      A     M    502.5;
      =     L      0.0;
      BLD   103;
      A     I    304.4;
      =     L      0.1;
      BLD   103;
      A     I    304.5;
      =     L      0.2;
      BLD   103;
      A     I    304.6;
      =     L      0.4;
      BLD   103;
      A     I    304.7;
      =     L      0.6;
      BLD   103;
      A     I    305.0;
      =     L      1.0;
      BLD   103;
      A     I    305.1;
      =     L      1.2;
      BLD   103;
      A     M    740.6;
      =     L      2.1;
      BLD   103;
      A     M    740.7;
      =     L      2.2;
      BLD   103;
      AN    M    504.0;
      AN    M    504.1;
      AN    M   6060.0;
      AN    M   6260.0;
      AN    M   6280.0;
      AN    M    504.2;
      A     M    500.2;
      =     L      2.3;
      BLD   103;
      A(    ;
      O     I      0.1;
      O     M   4120.1;
      )     ;
      =     L      2.5;
      BLD   103;
      A     M      0.5;
      =     L      2.6;
      BLD   103;
      CALL #S705_TL_DC_1ST_CLAMP1 (
           Enable_Aux               := L      0.0,
           Adv_Amount               := 1,
           Ret_Amount               := 5,
           LS_Adv1                  := L      0.1,
           LS_Ret1                  := L      0.2,
           LS_Ret2                  := L      0.4,
           LS_Ret3                  := L      0.6,
           LS_Ret4                  := L      1.0,
           LS_Ret5                  := L      1.2,
           SOL_Adv                  := L      2.1,
           SOL_Ret                  := L      2.2,
           M_Ready                  := L      2.3,
           T_CHK1                   := T#4S,
           T_CHK2                   := T#4S,
           PB_Error_Rst             := L      2.5,
           M_FLICK                  := L      2.6,
           M_Adv_Err                := M    750.6,
           M_Ret_Err                := M    750.7,
           Visu_Adv                 := DB51.DBW  132,
           Visu_Ret                 := DB51.DBW  134);
      NOP   0;
NETWORK
TITLE =
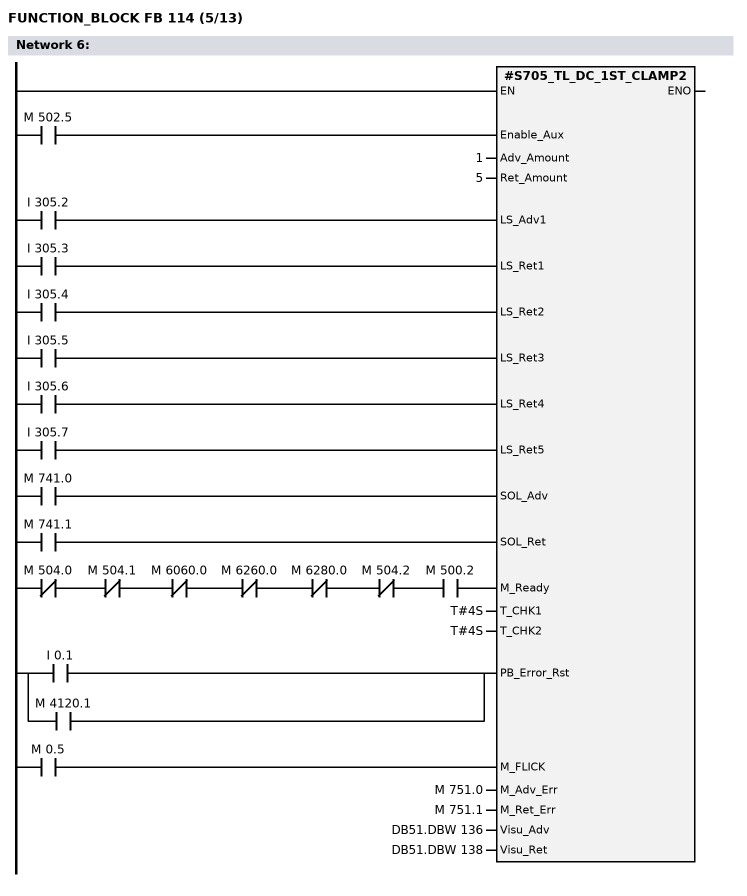

      A     M    502.5;
      =     L      0.0;
      BLD   103;
      A     I    305.2;
      =     L      0.1;
      BLD   103;
      A     I    305.3;
      =     L      0.2;
      BLD   103;
      A     I    305.4;
      =     L      0.4;
      BLD   103;
      A     I    305.5;
      =     L      0.6;
      BLD   103;
      A     I    305.6;
      =     L      1.0;
      BLD   103;
      A     I    305.7;
      =     L      1.2;
      BLD   103;
      A     M    741.0;
      =     L      2.1;
      BLD   103;
      A     M    741.1;
      =     L      2.2;
      BLD   103;
      AN    M    504.0;
      AN    M    504.1;
      AN    M   6060.0;
      AN    M   6260.0;
      AN    M   6280.0;
      AN    M    504.2;
      A     M    500.2;
      =     L      2.3;
      BLD   103;
      A(    ;
      O     I      0.1;
      O     M   4120.1;
      )     ;
      =     L      2.5;
      BLD   103;
      A     M      0.5;
      =     L      2.6;
      BLD   103;
      CALL #S705_TL_DC_1ST_CLAMP2 (
           Enable_Aux               := L      0.0,
           Adv_Amount               := 1,
           Ret_Amount               := 5,
           LS_Adv1                  := L      0.1,
           LS_Ret1                  := L      0.2,
           LS_Ret2                  := L      0.4,
           LS_Ret3                  := L      0.6,
           LS_Ret4                  := L      1.0,
           LS_Ret5                  := L      1.2,
           SOL_Adv                  := L      2.1,
           SOL_Ret                  := L      2.2,
           M_Ready                  := L      2.3,
           T_CHK1                   := T#4S,
           T_CHK2                   := T#4S,
           PB_Error_Rst             := L      2.5,
           M_FLICK                  := L      2.6,
           M_Adv_Err                := M    751.0,
           M_Ret_Err                := M    751.1,
           Visu_Adv                 := DB51.DBW  136,
           Visu_Ret                 := DB51.DBW  138);
      NOP   0;
NETWORK
TITLE =
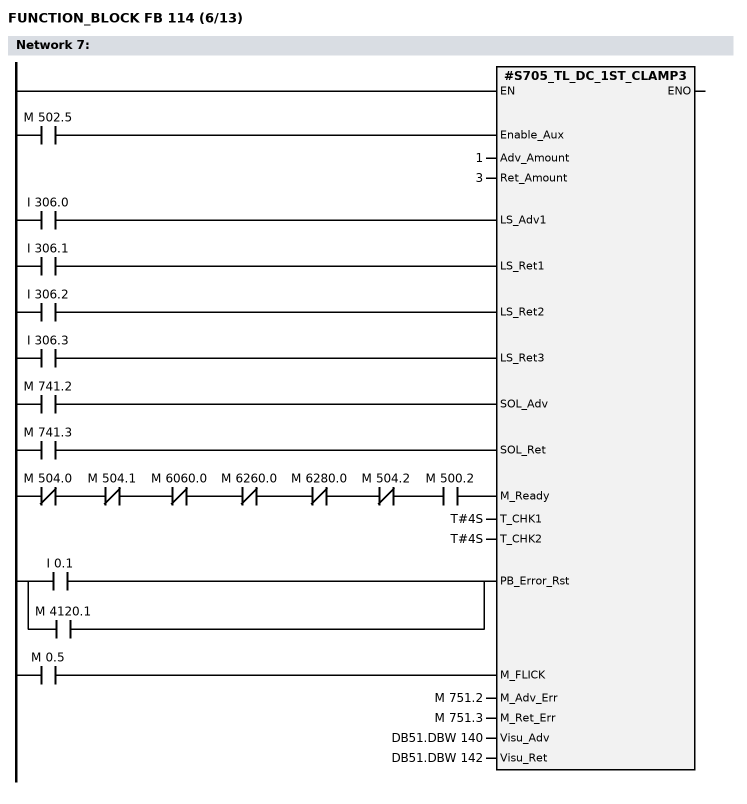

      A     M    502.5;
      =     L      0.0;
      BLD   103;
      A     I    306.0;
      =     L      0.1;
      BLD   103;
      A     I    306.1;
      =     L      0.2;
      BLD   103;
      A     I    306.2;
      =     L      0.4;
      BLD   103;
      A     I    306.3;
      =     L      0.6;
      BLD   103;
      A     M    741.2;
      =     L      2.1;
      BLD   103;
      A     M    741.3;
      =     L      2.2;
      BLD   103;
      AN    M    504.0;
      AN    M    504.1;
      AN    M   6060.0;
      AN    M   6260.0;
      AN    M   6280.0;
      AN    M    504.2;
      A     M    500.2;
      =     L      2.3;
      BLD   103;
      A(    ;
      O     I      0.1;
      O     M   4120.1;
      )     ;
      =     L      2.5;
      BLD   103;
      A     M      0.5;
      =     L      2.6;
      BLD   103;
      CALL #S705_TL_DC_1ST_CLAMP3 (
           Enable_Aux               := L      0.0,
           Adv_Amount               := 1,
           Ret_Amount               := 3,
           LS_Adv1                  := L      0.1,
           LS_Ret1                  := L      0.2,
           LS_Ret2                  := L      0.4,
           LS_Ret3                  := L      0.6,
           SOL_Adv                  := L      2.1,
           SOL_Ret                  := L      2.2,
           M_Ready                  := L      2.3,
           T_CHK1                   := T#4S,
           T_CHK2                   := T#4S,
           PB_Error_Rst             := L      2.5,
           M_FLICK                  := L      2.6,
           M_Adv_Err                := M    751.2,
           M_Ret_Err                := M    751.3,
           Visu_Adv                 := DB51.DBW  140,
           Visu_Ret                 := DB51.DBW  142);
      NOP   0;
NETWORK
TITLE =
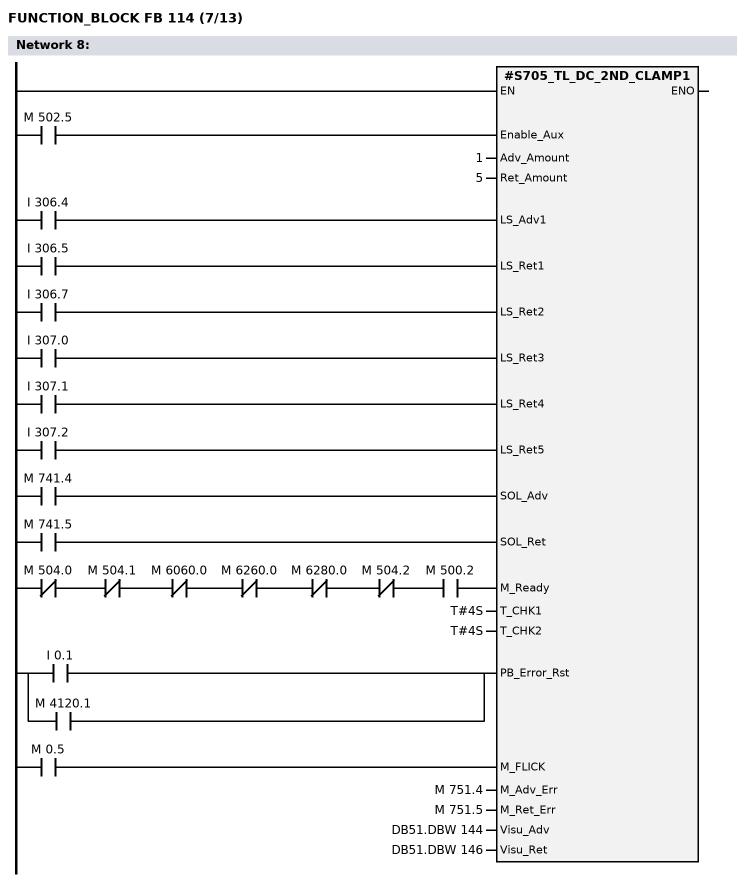

      A     M    502.5;
      =     L      0.0;
      BLD   103;
      A     I    306.4;
      =     L      0.1;
      BLD   103;
      A     I    306.5;
      =     L      0.2;
      BLD   103;
      A     I    306.7;
      =     L      0.4;
      BLD   103;
      A     I    307.0;
      =     L      0.6;
      BLD   103;
      A     I    307.1;
      =     L      1.0;
      BLD   103;
      A     I    307.2;
      =     L      1.2;
      BLD   103;
      A     M    741.4;
      =     L      2.1;
      BLD   103;
      A     M    741.5;
      =     L      2.2;
      BLD   103;
      AN    M    504.0;
      AN    M    504.1;
      AN    M   6060.0;
      AN    M   6260.0;
      AN    M   6280.0;
      AN    M    504.2;
      A     M    500.2;
      =     L      2.3;
      BLD   103;
      A(    ;
      O     I      0.1;
      O     M   4120.1;
      )     ;
      =     L      2.5;
      BLD   103;
      A     M      0.5;
      =     L      2.6;
      BLD   103;
      CALL #S705_TL_DC_2ND_CLAMP1 (
           Enable_Aux               := L      0.0,
           Adv_Amount               := 1,
           Ret_Amount               := 5,
           LS_Adv1                  := L      0.1,
           LS_Ret1                  := L      0.2,
           LS_Ret2                  := L      0.4,
           LS_Ret3                  := L      0.6,
           LS_Ret4                  := L      1.0,
           LS_Ret5                  := L      1.2,
           SOL_Adv                  := L      2.1,
           SOL_Ret                  := L      2.2,
           M_Ready                  := L      2.3,
           T_CHK1                   := T#4S,
           T_CHK2                   := T#4S,
           PB_Error_Rst             := L      2.5,
           M_FLICK                  := L      2.6,
           M_Adv_Err                := M    751.4,
           M_Ret_Err                := M    751.5,
           Visu_Adv                 := DB51.DBW  144,
           Visu_Ret                 := DB51.DBW  146);
      NOP   0;
NETWORK
TITLE =
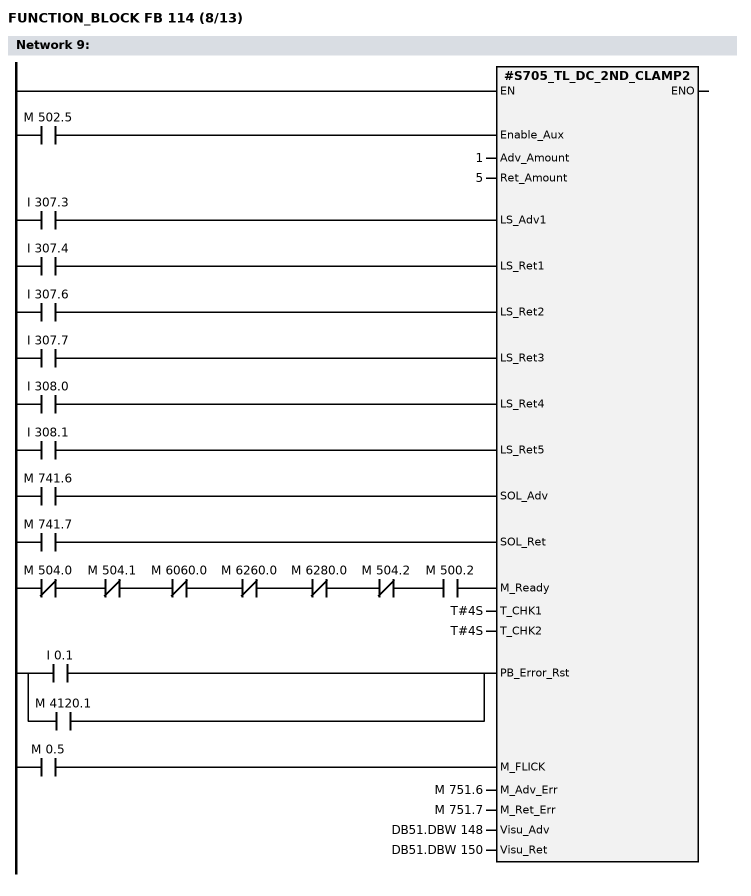

      A     M    502.5;
      =     L      0.0;
      BLD   103;
      A     I    307.3;
      =     L      0.1;
      BLD   103;
      A     I    307.4;
      =     L      0.2;
      BLD   103;
      A     I    307.6;
      =     L      0.4;
      BLD   103;
      A     I    307.7;
      =     L      0.6;
      BLD   103;
      A     I    308.0;
      =     L      1.0;
      BLD   103;
      A     I    308.1;
      =     L      1.2;
      BLD   103;
      A     M    741.6;
      =     L      2.1;
      BLD   103;
      A     M    741.7;
      =     L      2.2;
      BLD   103;
      AN    M    504.0;
      AN    M    504.1;
      AN    M   6060.0;
      AN    M   6260.0;
      AN    M   6280.0;
      AN    M    504.2;
      A     M    500.2;
      =     L      2.3;
      BLD   103;
      A(    ;
      O     I      0.1;
      O     M   4120.1;
      )     ;
      =     L      2.5;
      BLD   103;
      A     M      0.5;
      =     L      2.6;
      BLD   103;
      CALL #S705_TL_DC_2ND_CLAMP2 (
           Enable_Aux               := L      0.0,
           Adv_Amount               := 1,
           Ret_Amount               := 5,
           LS_Adv1                  := L      0.1,
           LS_Ret1                  := L      0.2,
           LS_Ret2                  := L      0.4,
           LS_Ret3                  := L      0.6,
           LS_Ret4                  := L      1.0,
           LS_Ret5                  := L      1.2,
           SOL_Adv                  := L      2.1,
           SOL_Ret                  := L      2.2,
           M_Ready                  := L      2.3,
           T_CHK1                   := T#4S,
           T_CHK2                   := T#4S,
           PB_Error_Rst             := L      2.5,
           M_FLICK                  := L      2.6,
           M_Adv_Err                := M    751.6,
           M_Ret_Err                := M    751.7,
           Visu_Adv                 := DB51.DBW  148,
           Visu_Ret                 := DB51.DBW  150);
      NOP   0;
NETWORK
TITLE =
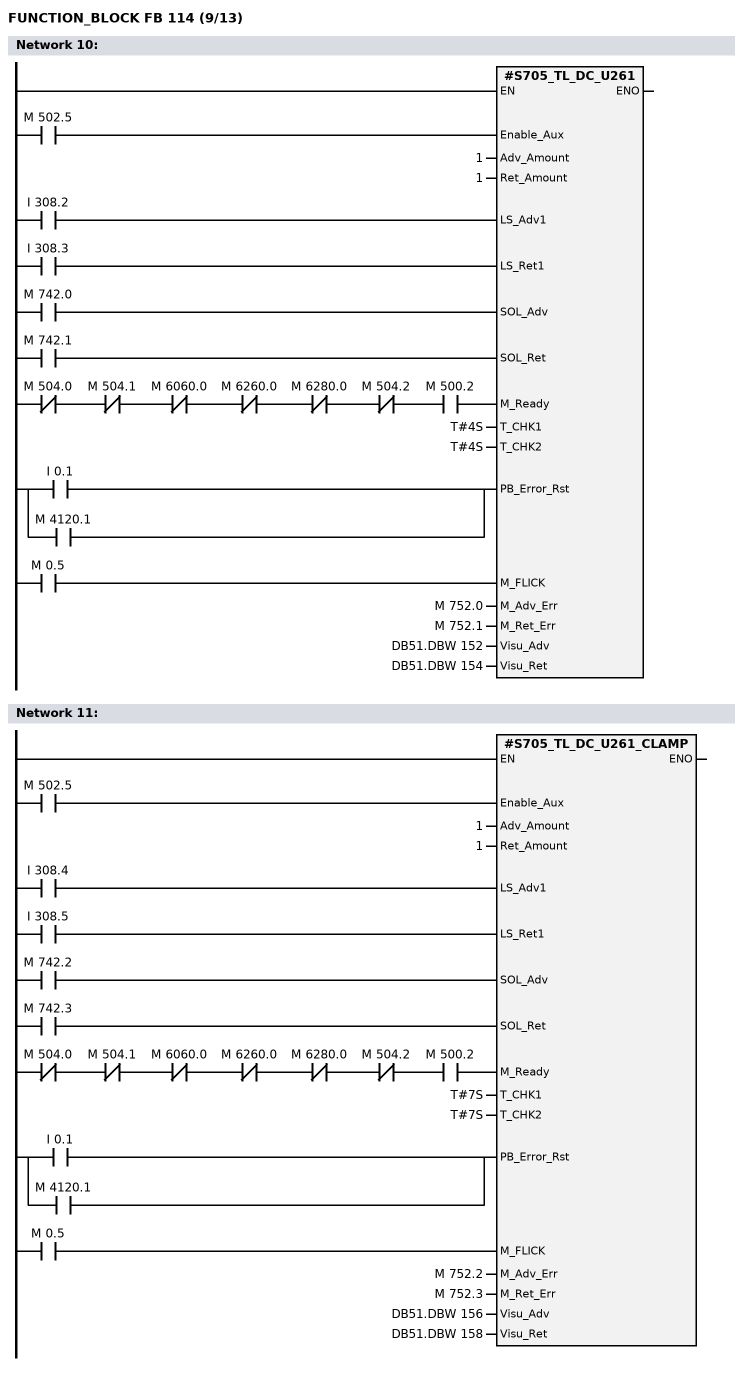

      A     M    502.5;
      =     L      0.0;
      BLD   103;
      A     I    308.2;
      =     L      0.1;
      BLD   103;
      A     I    308.3;
      =     L      0.2;
      BLD   103;
      A     M    742.0;
      =     L      2.1;
      BLD   103;
      A     M    742.1;
      =     L      2.2;
      BLD   103;
      AN    M    504.0;
      AN    M    504.1;
      AN    M   6060.0;
      AN    M   6260.0;
      AN    M   6280.0;
      AN    M    504.2;
      A     M    500.2;
      =     L      2.3;
      BLD   103;
      A(    ;
      O     I      0.1;
      O     M   4120.1;
      )     ;
      =     L      2.5;
      BLD   103;
      A     M      0.5;
      =     L      2.6;
      BLD   103;
      CALL #S705_TL_DC_U261 (
           Enable_Aux               := L      0.0,
           Adv_Amount               := 1,
           Ret_Amount               := 1,
           LS_Adv1                  := L      0.1,
           LS_Ret1                  := L      0.2,
           SOL_Adv                  := L      2.1,
           SOL_Ret                  := L      2.2,
           M_Ready                  := L      2.3,
           T_CHK1                   := T#4S,
           T_CHK2                   := T#4S,
           PB_Error_Rst             := L      2.5,
           M_FLICK                  := L      2.6,
           M_Adv_Err                := M    752.0,
           M_Ret_Err                := M    752.1,
           Visu_Adv                 := DB51.DBW  152,
           Visu_Ret                 := DB51.DBW  154);
      NOP   0;
NETWORK
TITLE =

      A     M    502.5;
      =     L      0.0;
      BLD   103;
      A     I    308.4;
      =     L      0.1;
      BLD   103;
      A     I    308.5;
      =     L      0.2;
      BLD   103;
      A     M    742.2;
      =     L      2.1;
      BLD   103;
      A     M    742.3;
      =     L      2.2;
      BLD   103;
      AN    M    504.0;
      AN    M    504.1;
      AN    M   6060.0;
      AN    M   6260.0;
      AN    M   6280.0;
      AN    M    504.2;
      A     M    500.2;
      =     L      2.3;
      BLD   103;
      A(    ;
      O     I      0.1;
      O     M   4120.1;
      )     ;
      =     L      2.5;
      BLD   103;
      A     M      0.5;
      =     L      2.6;
      BLD   103;
      CALL #S705_TL_DC_U261_CLAMP (
           Enable_Aux               := L      0.0,
           Adv_Amount               := 1,
           Ret_Amount               := 1,
           LS_Adv1                  := L      0.1,
           LS_Ret1                  := L      0.2,
           SOL_Adv                  := L      2.1,
           SOL_Ret                  := L      2.2,
           M_Ready                  := L      2.3,
           T_CHK1                   := T#7S,
           T_CHK2                   := T#7S,
           PB_Error_Rst             := L      2.5,
           M_FLICK                  := L      2.6,
           M_Adv_Err                := M    752.2,
           M_Ret_Err                := M    752.3,
           Visu_Adv                 := DB51.DBW  156,
           Visu_Ret                 := DB51.DBW  158);
      NOP   0;
NETWORK
TITLE =
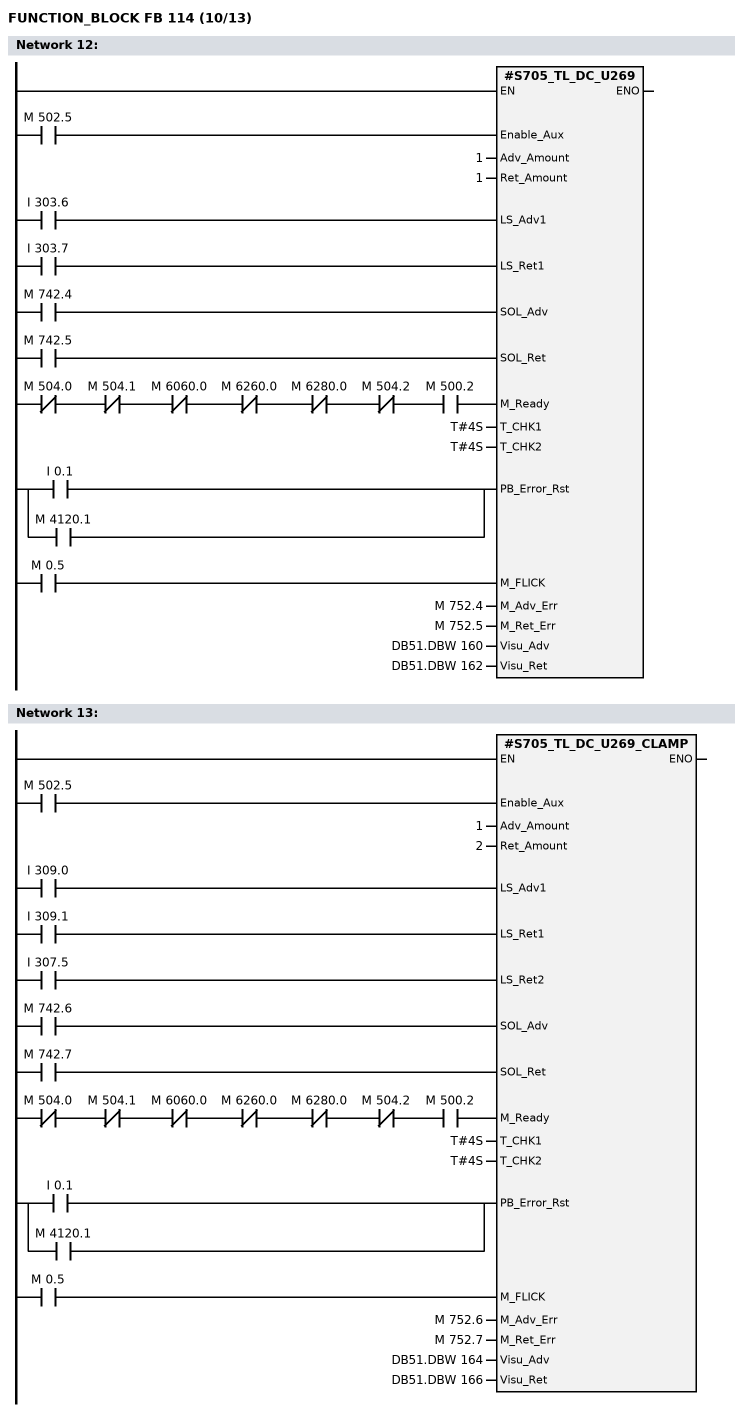

      A     M    502.5;
      =     L      0.0;
      BLD   103;
      A     I    303.6;
      =     L      0.1;
      BLD   103;
      A     I    303.7;
      =     L      0.2;
      BLD   103;
      A     M    742.4;
      =     L      2.1;
      BLD   103;
      A     M    742.5;
      =     L      2.2;
      BLD   103;
      AN    M    504.0;
      AN    M    504.1;
      AN    M   6060.0;
      AN    M   6260.0;
      AN    M   6280.0;
      AN    M    504.2;
      A     M    500.2;
      =     L      2.3;
      BLD   103;
      A(    ;
      O     I      0.1;
      O     M   4120.1;
      )     ;
      =     L      2.5;
      BLD   103;
      A     M      0.5;
      =     L      2.6;
      BLD   103;
      CALL #S705_TL_DC_U269 (
           Enable_Aux               := L      0.0,
           Adv_Amount               := 1,
           Ret_Amount               := 1,
           LS_Adv1                  := L      0.1,
           LS_Ret1                  := L      0.2,
           SOL_Adv                  := L      2.1,
           SOL_Ret                  := L      2.2,
           M_Ready                  := L      2.3,
           T_CHK1                   := T#4S,
           T_CHK2                   := T#4S,
           PB_Error_Rst             := L      2.5,
           M_FLICK                  := L      2.6,
           M_Adv_Err                := M    752.4,
           M_Ret_Err                := M    752.5,
           Visu_Adv                 := DB51.DBW  160,
           Visu_Ret                 := DB51.DBW  162);
      NOP   0;
NETWORK
TITLE =

      A     M    502.5;
      =     L      0.0;
      BLD   103;
      A     I    309.0;
      =     L      0.1;
      BLD   103;
      A     I    309.1;
      =     L      0.2;
      BLD   103;
      A     I    307.5;
      =     L      0.4;
      BLD   103;
      A     M    742.6;
      =     L      2.1;
      BLD   103;
      A     M    742.7;
      =     L      2.2;
      BLD   103;
      AN    M    504.0;
      AN    M    504.1;
      AN    M   6060.0;
      AN    M   6260.0;
      AN    M   6280.0;
      AN    M    504.2;
      A     M    500.2;
      =     L      2.3;
      BLD   103;
      A(    ;
      O     I      0.1;
      O     M   4120.1;
      )     ;
      =     L      2.5;
      BLD   103;
      A     M      0.5;
      =     L      2.6;
      BLD   103;
      CALL #S705_TL_DC_U269_CLAMP (
           Enable_Aux               := L      0.0,
           Adv_Amount               := 1,
           Ret_Amount               := 2,
           LS_Adv1                  := L      0.1,
           LS_Ret1                  := L      0.2,
           LS_Ret2                  := L      0.4,
           SOL_Adv                  := L      2.1,
           SOL_Ret                  := L      2.2,
           M_Ready                  := L      2.3,
           T_CHK1                   := T#4S,
           T_CHK2                   := T#4S,
           PB_Error_Rst             := L      2.5,
           M_FLICK                  := L      2.6,
           M_Adv_Err                := M    752.6,
           M_Ret_Err                := M    752.7,
           Visu_Adv                 := DB51.DBW  164,
           Visu_Ret                 := DB51.DBW  166);
      NOP   0;
NETWORK
TITLE =
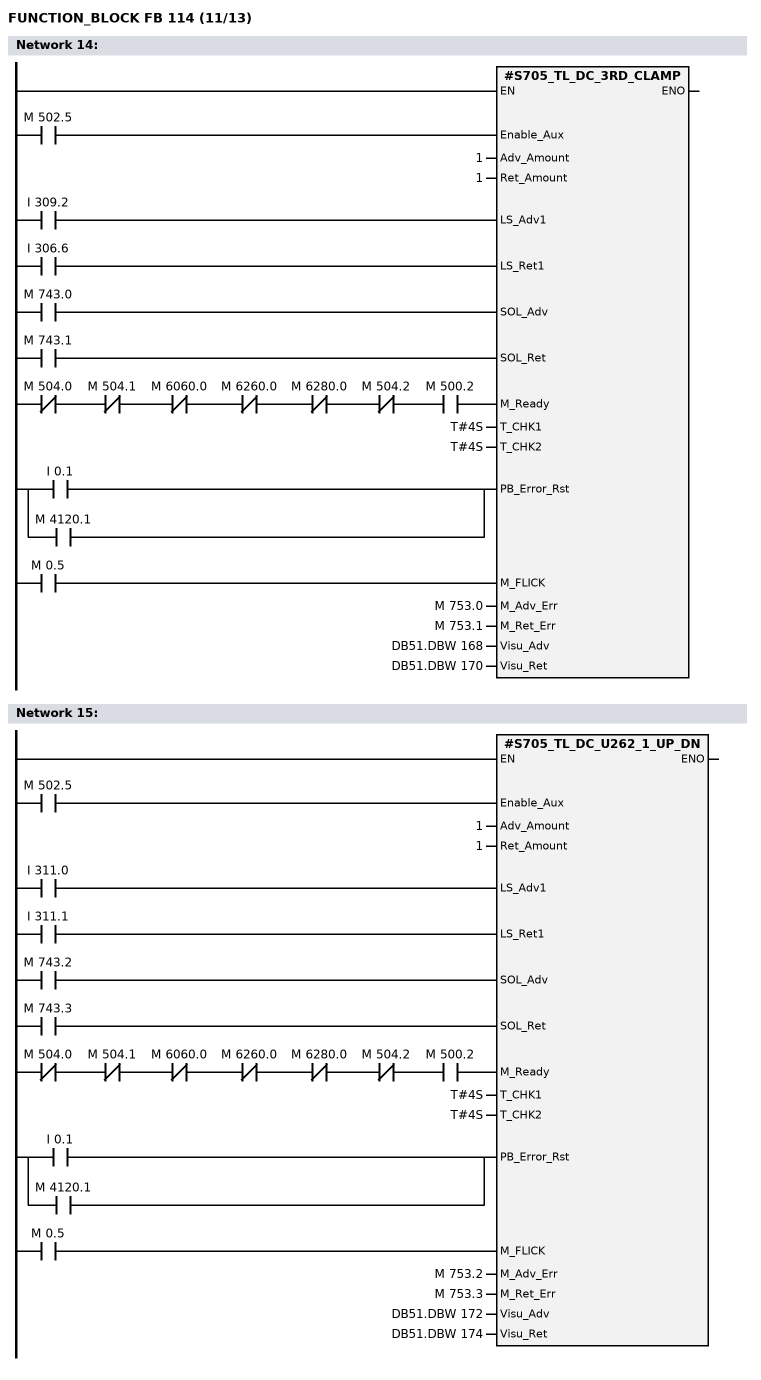

      A     M    502.5;
      =     L      0.0;
      BLD   103;
      A     I    309.2;
      =     L      0.1;
      BLD   103;
      A     I    306.6;
      =     L      0.2;
      BLD   103;
      A     M    743.0;
      =     L      2.1;
      BLD   103;
      A     M    743.1;
      =     L      2.2;
      BLD   103;
      AN    M    504.0;
      AN    M    504.1;
      AN    M   6060.0;
      AN    M   6260.0;
      AN    M   6280.0;
      AN    M    504.2;
      A     M    500.2;
      =     L      2.3;
      BLD   103;
      A(    ;
      O     I      0.1;
      O     M   4120.1;
      )     ;
      =     L      2.5;
      BLD   103;
      A     M      0.5;
      =     L      2.6;
      BLD   103;
      CALL #S705_TL_DC_3RD_CLAMP (
           Enable_Aux               := L      0.0,
           Adv_Amount               := 1,
           Ret_Amount               := 1,
           LS_Adv1                  := L      0.1,
           LS_Ret1                  := L      0.2,
           SOL_Adv                  := L      2.1,
           SOL_Ret                  := L      2.2,
           M_Ready                  := L      2.3,
           T_CHK1                   := T#4S,
           T_CHK2                   := T#4S,
           PB_Error_Rst             := L      2.5,
           M_FLICK                  := L      2.6,
           M_Adv_Err                := M    753.0,
           M_Ret_Err                := M    753.1,
           Visu_Adv                 := DB51.DBW  168,
           Visu_Ret                 := DB51.DBW  170);
      NOP   0;
NETWORK
TITLE =

      A     M    502.5;
      =     L      0.0;
      BLD   103;
      A     I    311.0;
      =     L      0.1;
      BLD   103;
      A     I    311.1;
      =     L      0.2;
      BLD   103;
      A     M    743.2;
      =     L      2.1;
      BLD   103;
      A     M    743.3;
      =     L      2.2;
      BLD   103;
      AN    M    504.0;
      AN    M    504.1;
      AN    M   6060.0;
      AN    M   6260.0;
      AN    M   6280.0;
      AN    M    504.2;
      A     M    500.2;
      =     L      2.3;
      BLD   103;
      A(    ;
      O     I      0.1;
      O     M   4120.1;
      )     ;
      =     L      2.5;
      BLD   103;
      A     M      0.5;
      =     L      2.6;
      BLD   103;
      CALL #S705_TL_DC_U262_1_UP_DN (
           Enable_Aux               := L      0.0,
           Adv_Amount               := 1,
           Ret_Amount               := 1,
           LS_Adv1                  := L      0.1,
           LS_Ret1                  := L      0.2,
           SOL_Adv                  := L      2.1,
           SOL_Ret                  := L      2.2,
           M_Ready                  := L      2.3,
           T_CHK1                   := T#4S,
           T_CHK2                   := T#4S,
           PB_Error_Rst             := L      2.5,
           M_FLICK                  := L      2.6,
           M_Adv_Err                := M    753.2,
           M_Ret_Err                := M    753.3,
           Visu_Adv                 := DB51.DBW  172,
           Visu_Ret                 := DB51.DBW  174);
      NOP   0;
NETWORK
TITLE =
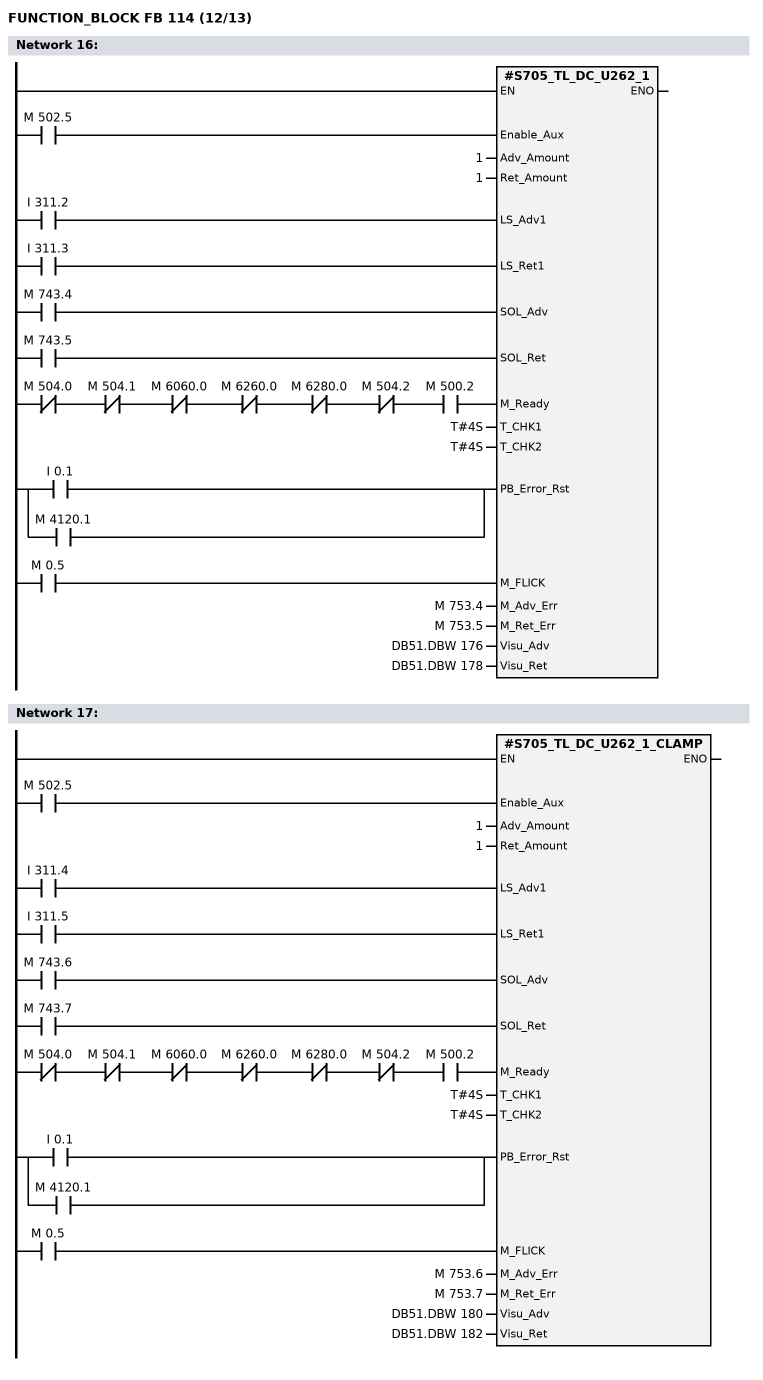

      A     M    502.5;
      =     L      0.0;
      BLD   103;
      A     I    311.2;
      =     L      0.1;
      BLD   103;
      A     I    311.3;
      =     L      0.2;
      BLD   103;
      A     M    743.4;
      =     L      2.1;
      BLD   103;
      A     M    743.5;
      =     L      2.2;
      BLD   103;
      AN    M    504.0;
      AN    M    504.1;
      AN    M   6060.0;
      AN    M   6260.0;
      AN    M   6280.0;
      AN    M    504.2;
      A     M    500.2;
      =     L      2.3;
      BLD   103;
      A(    ;
      O     I      0.1;
      O     M   4120.1;
      )     ;
      =     L      2.5;
      BLD   103;
      A     M      0.5;
      =     L      2.6;
      BLD   103;
      CALL #S705_TL_DC_U262_1 (
           Enable_Aux               := L      0.0,
           Adv_Amount               := 1,
           Ret_Amount               := 1,
           LS_Adv1                  := L      0.1,
           LS_Ret1                  := L      0.2,
           SOL_Adv                  := L      2.1,
           SOL_Ret                  := L      2.2,
           M_Ready                  := L      2.3,
           T_CHK1                   := T#4S,
           T_CHK2                   := T#4S,
           PB_Error_Rst             := L      2.5,
           M_FLICK                  := L      2.6,
           M_Adv_Err                := M    753.4,
           M_Ret_Err                := M    753.5,
           Visu_Adv                 := DB51.DBW  176,
           Visu_Ret                 := DB51.DBW  178);
      NOP   0;
NETWORK
TITLE =

      A     M    502.5;
      =     L      0.0;
      BLD   103;
      A     I    311.4;
      =     L      0.1;
      BLD   103;
      A     I    311.5;
      =     L      0.2;
      BLD   103;
      A     M    743.6;
      =     L      2.1;
      BLD   103;
      A     M    743.7;
      =     L      2.2;
      BLD   103;
      AN    M    504.0;
      AN    M    504.1;
      AN    M   6060.0;
      AN    M   6260.0;
      AN    M   6280.0;
      AN    M    504.2;
      A     M    500.2;
      =     L      2.3;
      BLD   103;
      A(    ;
      O     I      0.1;
      O     M   4120.1;
      )     ;
      =     L      2.5;
      BLD   103;
      A     M      0.5;
      =     L      2.6;
      BLD   103;
      CALL #S705_TL_DC_U262_1_CLAMP (
           Enable_Aux               := L      0.0,
           Adv_Amount               := 1,
           Ret_Amount               := 1,
           LS_Adv1                  := L      0.1,
           LS_Ret1                  := L      0.2,
           SOL_Adv                  := L      2.1,
           SOL_Ret                  := L      2.2,
           M_Ready                  := L      2.3,
           T_CHK1                   := T#4S,
           T_CHK2                   := T#4S,
           PB_Error_Rst             := L      2.5,
           M_FLICK                  := L      2.6,
           M_Adv_Err                := M    753.6,
           M_Ret_Err                := M    753.7,
           Visu_Adv                 := DB51.DBW  180,
           Visu_Ret                 := DB51.DBW  182);
      NOP   0;
NETWORK
TITLE =
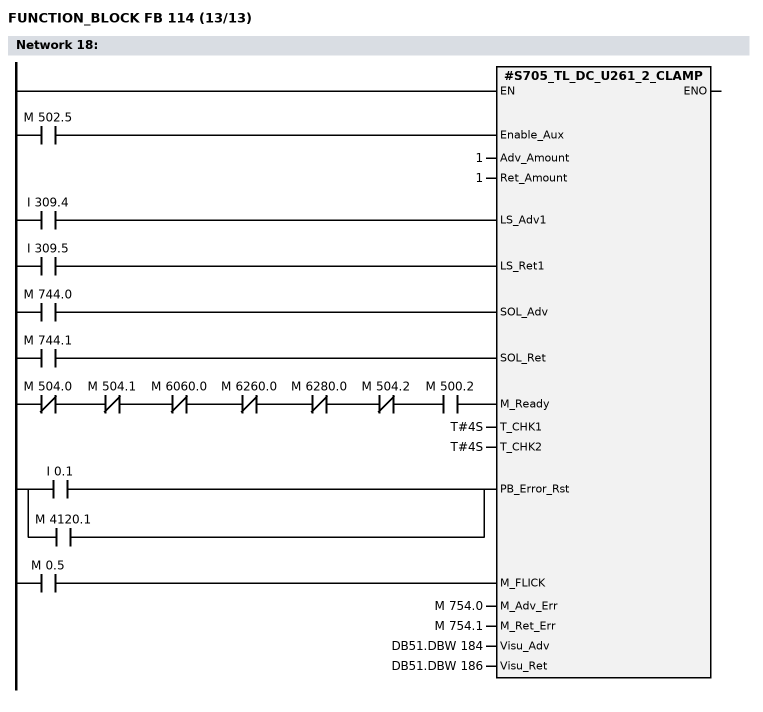

      A     M    502.5;
      =     L      0.0;
      BLD   103;
      A     I    309.4;
      =     L      0.1;
      BLD   103;
      A     I    309.5;
      =     L      0.2;
      BLD   103;
      A     M    744.0;
      =     L      2.1;
      BLD   103;
      A     M    744.1;
      =     L      2.2;
      BLD   103;
      AN    M    504.0;
      AN    M    504.1;
      AN    M   6060.0;
      AN    M   6260.0;
      AN    M   6280.0;
      AN    M    504.2;
      A     M    500.2;
      =     L      2.3;
      BLD   103;
      A(    ;
      O     I      0.1;
      O     M   4120.1;
      )     ;
      =     L      2.5;
      BLD   103;
      A     M      0.5;
      =     L      2.6;
      BLD   103;
      CALL #S705_TL_DC_U261_2_CLAMP (
           Enable_Aux               := L      0.0,
           Adv_Amount               := 1,
           Ret_Amount               := 1,
           LS_Adv1                  := L      0.1,
           LS_Ret1                  := L      0.2,
           SOL_Adv                  := L      2.1,
           SOL_Ret                  := L      2.2,
           M_Ready                  := L      2.3,
           T_CHK1                   := T#4S,
           T_CHK2                   := T#4S,
           PB_Error_Rst             := L      2.5,
           M_FLICK                  := L      2.6,
           M_Adv_Err                := M    754.0,
           M_Ret_Err                := M    754.1,
           Visu_Adv                 := DB51.DBW  184,
           Visu_Ret                 := DB51.DBW  186);
      NOP   0;
END_FUNCTION_BLOCK

DATA_BLOCK DB 114
TITLE =
VERSION : 0.0

 FB 114
BEGIN
   S705_TL_DC_PIN.Enable_Aux := TRUE;
   S705_TL_DC_PIN.Adv_Amount := 3;
   S705_TL_DC_PIN.Ret_Amount := 3;
   S705_TL_DC_PIN.LS_Adv1 := TRUE;
   S705_TL_DC_PIN.LS_Ret1 := FALSE;
   S705_TL_DC_PIN.LS_Adv2 := TRUE;
   S705_TL_DC_PIN.LS_Ret2 := FALSE;
   S705_TL_DC_PIN.LS_Adv3 := TRUE;
   S705_TL_DC_PIN.LS_Ret3 := FALSE;
   S705_TL_DC_PIN.LS_Adv4 := FALSE;
   S705_TL_DC_PIN.LS_Ret4 := FALSE;
   S705_TL_DC_PIN.LS_Adv5 := FALSE;
   S705_TL_DC_PIN.LS_Ret5 := FALSE;
   S705_TL_DC_PIN.LS_Adv6 := FALSE;
   S705_TL_DC_PIN.LS_Ret6 := FALSE;
   S705_TL_DC_PIN.LS_Adv7 := FALSE;
   S705_TL_DC_PIN.LS_Ret7 := FALSE;
   S705_TL_DC_PIN.LS_Adv8 := FALSE;
   S705_TL_DC_PIN.LS_Ret8 := FALSE;
   S705_TL_DC_PIN.SOL_Adv := FALSE;
   S705_TL_DC_PIN.SOL_Ret := FALSE;
   S705_TL_DC_PIN.M_Ready := TRUE;
   S705_TL_DC_PIN.T_CHK1 := T#4S;
   S705_TL_DC_PIN.T_CHK2 := T#4S;
   S705_TL_DC_PIN.PB_Lamp_CHK := FALSE;
   S705_TL_DC_PIN.PB_Error_Rst := FALSE;
   S705_TL_DC_PIN.M_FLICK := TRUE;
   S705_TL_DC_PIN.M_Adv_Err := FALSE;
   S705_TL_DC_PIN.M_Ret_Err := FALSE;
   S705_TL_DC_PIN.LP_Adv := TRUE;
   S705_TL_DC_PIN.LP_Ret := FALSE;
   S705_TL_DC_PIN.Visu_Adv := W#16#F00;
   S705_TL_DC_PIN.Visu_Ret := W#16#0;
   S705_TL_DC_PIN.Error_T1.IN := FALSE;
   S705_TL_DC_PIN.Error_T1.PT := T#4S;
   S705_TL_DC_PIN.Error_T1.Q := FALSE;
   S705_TL_DC_PIN.Error_T1.ET := T#0MS;
   S705_TL_DC_PIN.Error_T1.STATE := B#16#0;
   S705_TL_DC_PIN.Error_T1.STIME := T#23D3H47M22S548MS;
   S705_TL_DC_PIN.Error_T1.ATIME := T#23D3H47M22S592MS;
   S705_TL_DC_PIN.Error_T2.IN := FALSE;
   S705_TL_DC_PIN.Error_T2.PT := T#4S;
   S705_TL_DC_PIN.Error_T2.Q := FALSE;
   S705_TL_DC_PIN.Error_T2.ET := T#0MS;
   S705_TL_DC_PIN.Error_T2.STATE := B#16#0;
   S705_TL_DC_PIN.Error_T2.STIME := T#0MS;
   S705_TL_DC_PIN.Error_T2.ATIME := T#0MS;
   S705_TL_DC_PIN.Adv_End_Aux := TRUE;
   S705_TL_DC_PIN.Ret_End_Aux := FALSE;
   S705_TL_DC_PIN.CHK_Aux1 := FALSE;
   S705_TL_DC_PIN.CHK_Aux2 := FALSE;
   S705_TL_DC_PIN.Error_T1_DN := FALSE;
   S705_TL_DC_PIN.Error_T2_DN := FALSE;
   S705_TL_DC_PIN.Adv_Memo := TRUE;
   S705_TL_DC_PIN.Visu_Adv_Arr[0] := TRUE;
   S705_TL_DC_PIN.Visu_Adv_Arr[1] := TRUE;
   S705_TL_DC_PIN.Visu_Adv_Arr[2] := TRUE;
   S705_TL_DC_PIN.Visu_Adv_Arr[3] := TRUE;
   S705_TL_DC_PIN.Visu_Adv_Arr[4] := FALSE;
   S705_TL_DC_PIN.Visu_Adv_Arr[5] := FALSE;
   S705_TL_DC_PIN.Visu_Adv_Arr[6] := FALSE;
   S705_TL_DC_PIN.Visu_Adv_Arr[7] := FALSE;
   S705_TL_DC_PIN.Visu_Adv_Arr[8] := FALSE;
   S705_TL_DC_PIN.Visu_Adv_Arr[9] := FALSE;
   S705_TL_DC_PIN.Visu_Adv_Arr[10] := FALSE;
   S705_TL_DC_PIN.Visu_Adv_Arr[11] := FALSE;
   S705_TL_DC_PIN.Visu_Adv_Arr[12] := FALSE;
   S705_TL_DC_PIN.Visu_Adv_Arr[13] := FALSE;
   S705_TL_DC_PIN.Visu_Adv_Arr[14] := FALSE;
   S705_TL_DC_PIN.Visu_Adv_Arr[15] := FALSE;
   S705_TL_DC_PIN.Visu_Ret_Arr[0] := FALSE;
   S705_TL_DC_PIN.Visu_Ret_Arr[1] := FALSE;
   S705_TL_DC_PIN.Visu_Ret_Arr[2] := FALSE;
   S705_TL_DC_PIN.Visu_Ret_Arr[3] := FALSE;
   S705_TL_DC_PIN.Visu_Ret_Arr[4] := FALSE;
   S705_TL_DC_PIN.Visu_Ret_Arr[5] := FALSE;
   S705_TL_DC_PIN.Visu_Ret_Arr[6] := FALSE;
   S705_TL_DC_PIN.Visu_Ret_Arr[7] := FALSE;
   S705_TL_DC_PIN.Visu_Ret_Arr[8] := FALSE;
   S705_TL_DC_PIN.Visu_Ret_Arr[9] := FALSE;
   S705_TL_DC_PIN.Visu_Ret_Arr[10] := FALSE;
   S705_TL_DC_PIN.Visu_Ret_Arr[11] := FALSE;
   S705_TL_DC_PIN.Visu_Ret_Arr[12] := FALSE;
   S705_TL_DC_PIN.Visu_Ret_Arr[13] := FALSE;
   S705_TL_DC_PIN.Visu_Ret_Arr[14] := FALSE;
   S705_TL_DC_PIN.Visu_Ret_Arr[15] := FALSE;
   S705_TL_DC_PIN.BLK_Move_Ret := 0;
   S705_TL_DC_PIN.Enable := TRUE;
   S705_TL_DC_PIN.Adv_End := TRUE;
   S705_TL_DC_PIN.Ret_End := FALSE;
   S705_TL_DC_LATCH1.Enable_Aux := TRUE;
   S705_TL_DC_LATCH1.Adv_Amount := 5;
   S705_TL_DC_LATCH1.Ret_Amount := 5;
   S705_TL_DC_LATCH1.LS_Adv1 := FALSE;
   S705_TL_DC_LATCH1.LS_Ret1 := TRUE;
   S705_TL_DC_LATCH1.LS_Adv2 := FALSE;
   S705_TL_DC_LATCH1.LS_Ret2 := TRUE;
   S705_TL_DC_LATCH1.LS_Adv3 := FALSE;
   S705_TL_DC_LATCH1.LS_Ret3 := TRUE;
   S705_TL_DC_LATCH1.LS_Adv4 := FALSE;
   S705_TL_DC_LATCH1.LS_Ret4 := TRUE;
   S705_TL_DC_LATCH1.LS_Adv5 := FALSE;
   S705_TL_DC_LATCH1.LS_Ret5 := TRUE;
   S705_TL_DC_LATCH1.LS_Adv6 := FALSE;
   S705_TL_DC_LATCH1.LS_Ret6 := FALSE;
   S705_TL_DC_LATCH1.LS_Adv7 := FALSE;
   S705_TL_DC_LATCH1.LS_Ret7 := FALSE;
   S705_TL_DC_LATCH1.LS_Adv8 := FALSE;
   S705_TL_DC_LATCH1.LS_Ret8 := FALSE;
   S705_TL_DC_LATCH1.SOL_Adv := FALSE;
   S705_TL_DC_LATCH1.SOL_Ret := FALSE;
   S705_TL_DC_LATCH1.M_Ready := TRUE;
   S705_TL_DC_LATCH1.T_CHK1 := T#4S;
   S705_TL_DC_LATCH1.T_CHK2 := T#4S;
   S705_TL_DC_LATCH1.PB_Lamp_CHK := FALSE;
   S705_TL_DC_LATCH1.PB_Error_Rst := FALSE;
   S705_TL_DC_LATCH1.M_FLICK := TRUE;
   S705_TL_DC_LATCH1.M_Adv_Err := FALSE;
   S705_TL_DC_LATCH1.M_Ret_Err := FALSE;
   S705_TL_DC_LATCH1.LP_Adv := FALSE;
   S705_TL_DC_LATCH1.LP_Ret := TRUE;
   S705_TL_DC_LATCH1.Visu_Adv := W#16#0;
   S705_TL_DC_LATCH1.Visu_Ret := W#16#3F00;
   S705_TL_DC_LATCH1.Error_T1.IN := FALSE;
   S705_TL_DC_LATCH1.Error_T1.PT := T#4S;
   S705_TL_DC_LATCH1.Error_T1.Q := FALSE;
   S705_TL_DC_LATCH1.Error_T1.ET := T#0MS;
   S705_TL_DC_LATCH1.Error_T1.STATE := B#16#0;
   S705_TL_DC_LATCH1.Error_T1.STIME := T#23D5H8M50S203MS;
   S705_TL_DC_LATCH1.Error_T1.ATIME := T#23D5H8M51S620MS;
   S705_TL_DC_LATCH1.Error_T2.IN := FALSE;
   S705_TL_DC_LATCH1.Error_T2.PT := T#4S;
   S705_TL_DC_LATCH1.Error_T2.Q := FALSE;
   S705_TL_DC_LATCH1.Error_T2.ET := T#0MS;
   S705_TL_DC_LATCH1.Error_T2.STATE := B#16#0;
   S705_TL_DC_LATCH1.Error_T2.STIME := T#0MS;
   S705_TL_DC_LATCH1.Error_T2.ATIME := T#0MS;
   S705_TL_DC_LATCH1.Adv_End_Aux := FALSE;
   S705_TL_DC_LATCH1.Ret_End_Aux := TRUE;
   S705_TL_DC_LATCH1.CHK_Aux1 := FALSE;
   S705_TL_DC_LATCH1.CHK_Aux2 := FALSE;
   S705_TL_DC_LATCH1.Error_T1_DN := FALSE;
   S705_TL_DC_LATCH1.Error_T2_DN := FALSE;
   S705_TL_DC_LATCH1.Adv_Memo := FALSE;
   S705_TL_DC_LATCH1.Visu_Adv_Arr[0] := FALSE;
   S705_TL_DC_LATCH1.Visu_Adv_Arr[1] := FALSE;
   S705_TL_DC_LATCH1.Visu_Adv_Arr[2] := FALSE;
   S705_TL_DC_LATCH1.Visu_Adv_Arr[3] := FALSE;
   S705_TL_DC_LATCH1.Visu_Adv_Arr[4] := FALSE;
   S705_TL_DC_LATCH1.Visu_Adv_Arr[5] := FALSE;
   S705_TL_DC_LATCH1.Visu_Adv_Arr[6] := FALSE;
   S705_TL_DC_LATCH1.Visu_Adv_Arr[7] := FALSE;
   S705_TL_DC_LATCH1.Visu_Adv_Arr[8] := FALSE;
   S705_TL_DC_LATCH1.Visu_Adv_Arr[9] := FALSE;
   S705_TL_DC_LATCH1.Visu_Adv_Arr[10] := FALSE;
   S705_TL_DC_LATCH1.Visu_Adv_Arr[11] := FALSE;
   S705_TL_DC_LATCH1.Visu_Adv_Arr[12] := FALSE;
   S705_TL_DC_LATCH1.Visu_Adv_Arr[13] := FALSE;
   S705_TL_DC_LATCH1.Visu_Adv_Arr[14] := FALSE;
   S705_TL_DC_LATCH1.Visu_Adv_Arr[15] := FALSE;
   S705_TL_DC_LATCH1.Visu_Ret_Arr[0] := TRUE;
   S705_TL_DC_LATCH1.Visu_Ret_Arr[1] := TRUE;
   S705_TL_DC_LATCH1.Visu_Ret_Arr[2] := TRUE;
   S705_TL_DC_LATCH1.Visu_Ret_Arr[3] := TRUE;
   S705_TL_DC_LATCH1.Visu_Ret_Arr[4] := TRUE;
   S705_TL_DC_LATCH1.Visu_Ret_Arr[5] := TRUE;
   S705_TL_DC_LATCH1.Visu_Ret_Arr[6] := FALSE;
   S705_TL_DC_LATCH1.Visu_Ret_Arr[7] := FALSE;
   S705_TL_DC_LATCH1.Visu_Ret_Arr[8] := FALSE;
   S705_TL_DC_LATCH1.Visu_Ret_Arr[9] := FALSE;
   S705_TL_DC_LATCH1.Visu_Ret_Arr[10] := FALSE;
   S705_TL_DC_LATCH1.Visu_Ret_Arr[11] := FALSE;
   S705_TL_DC_LATCH1.Visu_Ret_Arr[12] := FALSE;
   S705_TL_DC_LATCH1.Visu_Ret_Arr[13] := FALSE;
   S705_TL_DC_LATCH1.Visu_Ret_Arr[14] := FALSE;
   S705_TL_DC_LATCH1.Visu_Ret_Arr[15] := FALSE;
   S705_TL_DC_LATCH1.BLK_Move_Ret := 0;
   S705_TL_DC_LATCH1.Enable := TRUE;
   S705_TL_DC_LATCH1.Adv_End := FALSE;
   S705_TL_DC_LATCH1.Ret_End := TRUE;
   S705_TL_DC_LATCH2.Enable_Aux := TRUE;
   S705_TL_DC_LATCH2.Adv_Amount := 2;
   S705_TL_DC_LATCH2.Ret_Amount := 2;
   S705_TL_DC_LATCH2.LS_Adv1 := FALSE;
   S705_TL_DC_LATCH2.LS_Ret1 := TRUE;
   S705_TL_DC_LATCH2.LS_Adv2 := FALSE;
   S705_TL_DC_LATCH2.LS_Ret2 := TRUE;
   S705_TL_DC_LATCH2.LS_Adv3 := FALSE;
   S705_TL_DC_LATCH2.LS_Ret3 := FALSE;
   S705_TL_DC_LATCH2.LS_Adv4 := FALSE;
   S705_TL_DC_LATCH2.LS_Ret4 := FALSE;
   S705_TL_DC_LATCH2.LS_Adv5 := FALSE;
   S705_TL_DC_LATCH2.LS_Ret5 := FALSE;
   S705_TL_DC_LATCH2.LS_Adv6 := FALSE;
   S705_TL_DC_LATCH2.LS_Ret6 := FALSE;
   S705_TL_DC_LATCH2.LS_Adv7 := FALSE;
   S705_TL_DC_LATCH2.LS_Ret7 := FALSE;
   S705_TL_DC_LATCH2.LS_Adv8 := FALSE;
   S705_TL_DC_LATCH2.LS_Ret8 := FALSE;
   S705_TL_DC_LATCH2.SOL_Adv := FALSE;
   S705_TL_DC_LATCH2.SOL_Ret := FALSE;
   S705_TL_DC_LATCH2.M_Ready := TRUE;
   S705_TL_DC_LATCH2.T_CHK1 := T#4S;
   S705_TL_DC_LATCH2.T_CHK2 := T#4S;
   S705_TL_DC_LATCH2.PB_Lamp_CHK := FALSE;
   S705_TL_DC_LATCH2.PB_Error_Rst := FALSE;
   S705_TL_DC_LATCH2.M_FLICK := TRUE;
   S705_TL_DC_LATCH2.M_Adv_Err := FALSE;
   S705_TL_DC_LATCH2.M_Ret_Err := FALSE;
   S705_TL_DC_LATCH2.LP_Adv := FALSE;
   S705_TL_DC_LATCH2.LP_Ret := TRUE;
   S705_TL_DC_LATCH2.Visu_Adv := W#16#0;
   S705_TL_DC_LATCH2.Visu_Ret := W#16#100;
   S705_TL_DC_LATCH2.Error_T1.IN := FALSE;
   S705_TL_DC_LATCH2.Error_T1.PT := T#4S;
   S705_TL_DC_LATCH2.Error_T1.Q := FALSE;
   S705_TL_DC_LATCH2.Error_T1.ET := T#0MS;
   S705_TL_DC_LATCH2.Error_T1.STATE := B#16#0;
   S705_TL_DC_LATCH2.Error_T1.STIME := T#23D5H8M46S915MS;
   S705_TL_DC_LATCH2.Error_T1.ATIME := T#23D5H8M46S961MS;
   S705_TL_DC_LATCH2.Error_T2.IN := FALSE;
   S705_TL_DC_LATCH2.Error_T2.PT := T#4S;
   S705_TL_DC_LATCH2.Error_T2.Q := FALSE;
   S705_TL_DC_LATCH2.Error_T2.ET := T#0MS;
   S705_TL_DC_LATCH2.Error_T2.STATE := B#16#0;
   S705_TL_DC_LATCH2.Error_T2.STIME := T#0MS;
   S705_TL_DC_LATCH2.Error_T2.ATIME := T#0MS;
   S705_TL_DC_LATCH2.Adv_End_Aux := FALSE;
   S705_TL_DC_LATCH2.Ret_End_Aux := TRUE;
   S705_TL_DC_LATCH2.CHK_Aux1 := FALSE;
   S705_TL_DC_LATCH2.CHK_Aux2 := FALSE;
   S705_TL_DC_LATCH2.Error_T1_DN := FALSE;
   S705_TL_DC_LATCH2.Error_T2_DN := FALSE;
   S705_TL_DC_LATCH2.Adv_Memo := TRUE;
   S705_TL_DC_LATCH2.Visu_Adv_Arr[0] := FALSE;
   S705_TL_DC_LATCH2.Visu_Adv_Arr[1] := FALSE;
   S705_TL_DC_LATCH2.Visu_Adv_Arr[2] := FALSE;
   S705_TL_DC_LATCH2.Visu_Adv_Arr[3] := FALSE;
   S705_TL_DC_LATCH2.Visu_Adv_Arr[4] := FALSE;
   S705_TL_DC_LATCH2.Visu_Adv_Arr[5] := FALSE;
   S705_TL_DC_LATCH2.Visu_Adv_Arr[6] := FALSE;
   S705_TL_DC_LATCH2.Visu_Adv_Arr[7] := FALSE;
   S705_TL_DC_LATCH2.Visu_Adv_Arr[8] := FALSE;
   S705_TL_DC_LATCH2.Visu_Adv_Arr[9] := FALSE;
   S705_TL_DC_LATCH2.Visu_Adv_Arr[10] := FALSE;
   S705_TL_DC_LATCH2.Visu_Adv_Arr[11] := FALSE;
   S705_TL_DC_LATCH2.Visu_Adv_Arr[12] := FALSE;
   S705_TL_DC_LATCH2.Visu_Adv_Arr[13] := FALSE;
   S705_TL_DC_LATCH2.Visu_Adv_Arr[14] := FALSE;
   S705_TL_DC_LATCH2.Visu_Adv_Arr[15] := FALSE;
   S705_TL_DC_LATCH2.Visu_Ret_Arr[0] := TRUE;
   S705_TL_DC_LATCH2.Visu_Ret_Arr[1] := FALSE;
   S705_TL_DC_LATCH2.Visu_Ret_Arr[2] := FALSE;
   S705_TL_DC_LATCH2.Visu_Ret_Arr[3] := FALSE;
   S705_TL_DC_LATCH2.Visu_Ret_Arr[4] := FALSE;
   S705_TL_DC_LATCH2.Visu_Ret_Arr[5] := FALSE;
   S705_TL_DC_LATCH2.Visu_Ret_Arr[6] := FALSE;
   S705_TL_DC_LATCH2.Visu_Ret_Arr[7] := FALSE;
   S705_TL_DC_LATCH2.Visu_Ret_Arr[8] := FALSE;
   S705_TL_DC_LATCH2.Visu_Ret_Arr[9] := FALSE;
   S705_TL_DC_LATCH2.Visu_Ret_Arr[10] := FALSE;
   S705_TL_DC_LATCH2.Visu_Ret_Arr[11] := FALSE;
   S705_TL_DC_LATCH2.Visu_Ret_Arr[12] := FALSE;
   S705_TL_DC_LATCH2.Visu_Ret_Arr[13] := FALSE;
   S705_TL_DC_LATCH2.Visu_Ret_Arr[14] := FALSE;
   S705_TL_DC_LATCH2.Visu_Ret_Arr[15] := FALSE;
   S705_TL_DC_LATCH2.BLK_Move_Ret := 0;
   S705_TL_DC_LATCH2.Enable := TRUE;
   S705_TL_DC_LATCH2.Adv_End := FALSE;
   S705_TL_DC_LATCH2.Ret_End := TRUE;
   S705_TL_DC_1ST_CLAMP1.Enable_Aux := TRUE;
   S705_TL_DC_1ST_CLAMP1.Adv_Amount := 1;
   S705_TL_DC_1ST_CLAMP1.Ret_Amount := 5;
   S705_TL_DC_1ST_CLAMP1.LS_Adv1 := FALSE;
   S705_TL_DC_1ST_CLAMP1.LS_Ret1 := TRUE;
   S705_TL_DC_1ST_CLAMP1.LS_Adv2 := FALSE;
   S705_TL_DC_1ST_CLAMP1.LS_Ret2 := TRUE;
   S705_TL_DC_1ST_CLAMP1.LS_Adv3 := FALSE;
   S705_TL_DC_1ST_CLAMP1.LS_Ret3 := TRUE;
   S705_TL_DC_1ST_CLAMP1.LS_Adv4 := FALSE;
   S705_TL_DC_1ST_CLAMP1.LS_Ret4 := TRUE;
   S705_TL_DC_1ST_CLAMP1.LS_Adv5 := FALSE;
   S705_TL_DC_1ST_CLAMP1.LS_Ret5 := TRUE;
   S705_TL_DC_1ST_CLAMP1.LS_Adv6 := FALSE;
   S705_TL_DC_1ST_CLAMP1.LS_Ret6 := FALSE;
   S705_TL_DC_1ST_CLAMP1.LS_Adv7 := FALSE;
   S705_TL_DC_1ST_CLAMP1.LS_Ret7 := FALSE;
   S705_TL_DC_1ST_CLAMP1.LS_Adv8 := FALSE;
   S705_TL_DC_1ST_CLAMP1.LS_Ret8 := FALSE;
   S705_TL_DC_1ST_CLAMP1.SOL_Adv := FALSE;
   S705_TL_DC_1ST_CLAMP1.SOL_Ret := FALSE;
   S705_TL_DC_1ST_CLAMP1.M_Ready := TRUE;
   S705_TL_DC_1ST_CLAMP1.T_CHK1 := T#4S;
   S705_TL_DC_1ST_CLAMP1.T_CHK2 := T#4S;
   S705_TL_DC_1ST_CLAMP1.PB_Lamp_CHK := FALSE;
   S705_TL_DC_1ST_CLAMP1.PB_Error_Rst := FALSE;
   S705_TL_DC_1ST_CLAMP1.M_FLICK := TRUE;
   S705_TL_DC_1ST_CLAMP1.M_Adv_Err := FALSE;
   S705_TL_DC_1ST_CLAMP1.M_Ret_Err := FALSE;
   S705_TL_DC_1ST_CLAMP1.LP_Adv := FALSE;
   S705_TL_DC_1ST_CLAMP1.LP_Ret := TRUE;
   S705_TL_DC_1ST_CLAMP1.Visu_Adv := W#16#0;
   S705_TL_DC_1ST_CLAMP1.Visu_Ret := W#16#3F00;
   S705_TL_DC_1ST_CLAMP1.Error_T1.IN := FALSE;
   S705_TL_DC_1ST_CLAMP1.Error_T1.PT := T#4S;
   S705_TL_DC_1ST_CLAMP1.Error_T1.Q := FALSE;
   S705_TL_DC_1ST_CLAMP1.Error_T1.ET := T#0MS;
   S705_TL_DC_1ST_CLAMP1.Error_T1.STATE := B#16#0;
   S705_TL_DC_1ST_CLAMP1.Error_T1.STIME := T#23D5H8M48S571MS;
   S705_TL_DC_1ST_CLAMP1.Error_T1.ATIME := T#23D5H8M50S203MS;
   S705_TL_DC_1ST_CLAMP1.Error_T2.IN := FALSE;
   S705_TL_DC_1ST_CLAMP1.Error_T2.PT := T#4S;
   S705_TL_DC_1ST_CLAMP1.Error_T2.Q := FALSE;
   S705_TL_DC_1ST_CLAMP1.Error_T2.ET := T#0MS;
   S705_TL_DC_1ST_CLAMP1.Error_T2.STATE := B#16#0;
   S705_TL_DC_1ST_CLAMP1.Error_T2.STIME := T#0MS;
   S705_TL_DC_1ST_CLAMP1.Error_T2.ATIME := T#0MS;
   S705_TL_DC_1ST_CLAMP1.Adv_End_Aux := FALSE;
   S705_TL_DC_1ST_CLAMP1.Ret_End_Aux := TRUE;
   S705_TL_DC_1ST_CLAMP1.CHK_Aux1 := FALSE;
   S705_TL_DC_1ST_CLAMP1.CHK_Aux2 := FALSE;
   S705_TL_DC_1ST_CLAMP1.Error_T1_DN := FALSE;
   S705_TL_DC_1ST_CLAMP1.Error_T2_DN := FALSE;
   S705_TL_DC_1ST_CLAMP1.Adv_Memo := FALSE;
   S705_TL_DC_1ST_CLAMP1.Visu_Adv_Arr[0] := FALSE;
   S705_TL_DC_1ST_CLAMP1.Visu_Adv_Arr[1] := FALSE;
   S705_TL_DC_1ST_CLAMP1.Visu_Adv_Arr[2] := FALSE;
   S705_TL_DC_1ST_CLAMP1.Visu_Adv_Arr[3] := FALSE;
   S705_TL_DC_1ST_CLAMP1.Visu_Adv_Arr[4] := FALSE;
   S705_TL_DC_1ST_CLAMP1.Visu_Adv_Arr[5] := FALSE;
   S705_TL_DC_1ST_CLAMP1.Visu_Adv_Arr[6] := FALSE;
   S705_TL_DC_1ST_CLAMP1.Visu_Adv_Arr[7] := FALSE;
   S705_TL_DC_1ST_CLAMP1.Visu_Adv_Arr[8] := FALSE;
   S705_TL_DC_1ST_CLAMP1.Visu_Adv_Arr[9] := FALSE;
   S705_TL_DC_1ST_CLAMP1.Visu_Adv_Arr[10] := FALSE;
   S705_TL_DC_1ST_CLAMP1.Visu_Adv_Arr[11] := FALSE;
   S705_TL_DC_1ST_CLAMP1.Visu_Adv_Arr[12] := FALSE;
   S705_TL_DC_1ST_CLAMP1.Visu_Adv_Arr[13] := FALSE;
   S705_TL_DC_1ST_CLAMP1.Visu_Adv_Arr[14] := FALSE;
   S705_TL_DC_1ST_CLAMP1.Visu_Adv_Arr[15] := FALSE;
   S705_TL_DC_1ST_CLAMP1.Visu_Ret_Arr[0] := TRUE;
   S705_TL_DC_1ST_CLAMP1.Visu_Ret_Arr[1] := TRUE;
   S705_TL_DC_1ST_CLAMP1.Visu_Ret_Arr[2] := TRUE;
   S705_TL_DC_1ST_CLAMP1.Visu_Ret_Arr[3] := TRUE;
   S705_TL_DC_1ST_CLAMP1.Visu_Ret_Arr[4] := TRUE;
   S705_TL_DC_1ST_CLAMP1.Visu_Ret_Arr[5] := TRUE;
   S705_TL_DC_1ST_CLAMP1.Visu_Ret_Arr[6] := FALSE;
   S705_TL_DC_1ST_CLAMP1.Visu_Ret_Arr[7] := FALSE;
   S705_TL_DC_1ST_CLAMP1.Visu_Ret_Arr[8] := FALSE;
   S705_TL_DC_1ST_CLAMP1.Visu_Ret_Arr[9] := FALSE;
   S705_TL_DC_1ST_CLAMP1.Visu_Ret_Arr[10] := FALSE;
   S705_TL_DC_1ST_CLAMP1.Visu_Ret_Arr[11] := FALSE;
   S705_TL_DC_1ST_CLAMP1.Visu_Ret_Arr[12] := FALSE;
   S705_TL_DC_1ST_CLAMP1.Visu_Ret_Arr[13] := FALSE;
   S705_TL_DC_1ST_CLAMP1.Visu_Ret_Arr[14] := FALSE;
   S705_TL_DC_1ST_CLAMP1.Visu_Ret_Arr[15] := FALSE;
   S705_TL_DC_1ST_CLAMP1.BLK_Move_Ret := 0;
   S705_TL_DC_1ST_CLAMP1.Enable := TRUE;
   S705_TL_DC_1ST_CLAMP1.Adv_End := FALSE;
   S705_TL_DC_1ST_CLAMP1.Ret_End := TRUE;
   S705_TL_DC_1ST_CLAMP2.Enable_Aux := TRUE;
   S705_TL_DC_1ST_CLAMP2.Adv_Amount := 1;
   S705_TL_DC_1ST_CLAMP2.Ret_Amount := 5;
   S705_TL_DC_1ST_CLAMP2.LS_Adv1 := FALSE;
   S705_TL_DC_1ST_CLAMP2.LS_Ret1 := TRUE;
   S705_TL_DC_1ST_CLAMP2.LS_Adv2 := FALSE;
   S705_TL_DC_1ST_CLAMP2.LS_Ret2 := TRUE;
   S705_TL_DC_1ST_CLAMP2.LS_Adv3 := FALSE;
   S705_TL_DC_1ST_CLAMP2.LS_Ret3 := TRUE;
   S705_TL_DC_1ST_CLAMP2.LS_Adv4 := FALSE;
   S705_TL_DC_1ST_CLAMP2.LS_Ret4 := TRUE;
   S705_TL_DC_1ST_CLAMP2.LS_Adv5 := FALSE;
   S705_TL_DC_1ST_CLAMP2.LS_Ret5 := TRUE;
   S705_TL_DC_1ST_CLAMP2.LS_Adv6 := FALSE;
   S705_TL_DC_1ST_CLAMP2.LS_Ret6 := FALSE;
   S705_TL_DC_1ST_CLAMP2.LS_Adv7 := FALSE;
   S705_TL_DC_1ST_CLAMP2.LS_Ret7 := FALSE;
   S705_TL_DC_1ST_CLAMP2.LS_Adv8 := FALSE;
   S705_TL_DC_1ST_CLAMP2.LS_Ret8 := FALSE;
   S705_TL_DC_1ST_CLAMP2.SOL_Adv := FALSE;
   S705_TL_DC_1ST_CLAMP2.SOL_Ret := FALSE;
   S705_TL_DC_1ST_CLAMP2.M_Ready := TRUE;
   S705_TL_DC_1ST_CLAMP2.T_CHK1 := T#4S;
   S705_TL_DC_1ST_CLAMP2.T_CHK2 := T#4S;
   S705_TL_DC_1ST_CLAMP2.PB_Lamp_CHK := FALSE;
   S705_TL_DC_1ST_CLAMP2.PB_Error_Rst := FALSE;
   S705_TL_DC_1ST_CLAMP2.M_FLICK := TRUE;
   S705_TL_DC_1ST_CLAMP2.M_Adv_Err := FALSE;
   S705_TL_DC_1ST_CLAMP2.M_Ret_Err := FALSE;
   S705_TL_DC_1ST_CLAMP2.LP_Adv := FALSE;
   S705_TL_DC_1ST_CLAMP2.LP_Ret := TRUE;
   S705_TL_DC_1ST_CLAMP2.Visu_Adv := W#16#0;
   S705_TL_DC_1ST_CLAMP2.Visu_Ret := W#16#3F00;
   S705_TL_DC_1ST_CLAMP2.Error_T1.IN := FALSE;
   S705_TL_DC_1ST_CLAMP2.Error_T1.PT := T#4S;
   S705_TL_DC_1ST_CLAMP2.Error_T1.Q := FALSE;
   S705_TL_DC_1ST_CLAMP2.Error_T1.ET := T#0MS;
   S705_TL_DC_1ST_CLAMP2.Error_T1.STATE := B#16#0;
   S705_TL_DC_1ST_CLAMP2.Error_T1.STIME := T#23D5H8M48S572MS;
   S705_TL_DC_1ST_CLAMP2.Error_T1.ATIME := T#23D5H8M49S652MS;
   S705_TL_DC_1ST_CLAMP2.Error_T2.IN := FALSE;
   S705_TL_DC_1ST_CLAMP2.Error_T2.PT := T#4S;
   S705_TL_DC_1ST_CLAMP2.Error_T2.Q := FALSE;
   S705_TL_DC_1ST_CLAMP2.Error_T2.ET := T#0MS;
   S705_TL_DC_1ST_CLAMP2.Error_T2.STATE := B#16#0;
   S705_TL_DC_1ST_CLAMP2.Error_T2.STIME := T#0MS;
   S705_TL_DC_1ST_CLAMP2.Error_T2.ATIME := T#0MS;
   S705_TL_DC_1ST_CLAMP2.Adv_End_Aux := FALSE;
   S705_TL_DC_1ST_CLAMP2.Ret_End_Aux := TRUE;
   S705_TL_DC_1ST_CLAMP2.CHK_Aux1 := FALSE;
   S705_TL_DC_1ST_CLAMP2.CHK_Aux2 := FALSE;
   S705_TL_DC_1ST_CLAMP2.Error_T1_DN := FALSE;
   S705_TL_DC_1ST_CLAMP2.Error_T2_DN := FALSE;
   S705_TL_DC_1ST_CLAMP2.Adv_Memo := FALSE;
   S705_TL_DC_1ST_CLAMP2.Visu_Adv_Arr[0] := FALSE;
   S705_TL_DC_1ST_CLAMP2.Visu_Adv_Arr[1] := FALSE;
   S705_TL_DC_1ST_CLAMP2.Visu_Adv_Arr[2] := FALSE;
   S705_TL_DC_1ST_CLAMP2.Visu_Adv_Arr[3] := FALSE;
   S705_TL_DC_1ST_CLAMP2.Visu_Adv_Arr[4] := FALSE;
   S705_TL_DC_1ST_CLAMP2.Visu_Adv_Arr[5] := FALSE;
   S705_TL_DC_1ST_CLAMP2.Visu_Adv_Arr[6] := FALSE;
   S705_TL_DC_1ST_CLAMP2.Visu_Adv_Arr[7] := FALSE;
   S705_TL_DC_1ST_CLAMP2.Visu_Adv_Arr[8] := FALSE;
   S705_TL_DC_1ST_CLAMP2.Visu_Adv_Arr[9] := FALSE;
   S705_TL_DC_1ST_CLAMP2.Visu_Adv_Arr[10] := FALSE;
   S705_TL_DC_1ST_CLAMP2.Visu_Adv_Arr[11] := FALSE;
   S705_TL_DC_1ST_CLAMP2.Visu_Adv_Arr[12] := FALSE;
   S705_TL_DC_1ST_CLAMP2.Visu_Adv_Arr[13] := FALSE;
   S705_TL_DC_1ST_CLAMP2.Visu_Adv_Arr[14] := FALSE;
   S705_TL_DC_1ST_CLAMP2.Visu_Adv_Arr[15] := FALSE;
   S705_TL_DC_1ST_CLAMP2.Visu_Ret_Arr[0] := TRUE;
   S705_TL_DC_1ST_CLAMP2.Visu_Ret_Arr[1] := TRUE;
   S705_TL_DC_1ST_CLAMP2.Visu_Ret_Arr[2] := TRUE;
   S705_TL_DC_1ST_CLAMP2.Visu_Ret_Arr[3] := TRUE;
   S705_TL_DC_1ST_CLAMP2.Visu_Ret_Arr[4] := TRUE;
   S705_TL_DC_1ST_CLAMP2.Visu_Ret_Arr[5] := TRUE;
   S705_TL_DC_1ST_CLAMP2.Visu_Ret_Arr[6] := FALSE;
   S705_TL_DC_1ST_CLAMP2.Visu_Ret_Arr[7] := FALSE;
   S705_TL_DC_1ST_CLAMP2.Visu_Ret_Arr[8] := FALSE;
   S705_TL_DC_1ST_CLAMP2.Visu_Ret_Arr[9] := FALSE;
   S705_TL_DC_1ST_CLAMP2.Visu_Ret_Arr[10] := FALSE;
   S705_TL_DC_1ST_CLAMP2.Visu_Ret_Arr[11] := FALSE;
   S705_TL_DC_1ST_CLAMP2.Visu_Ret_Arr[12] := FALSE;
   S705_TL_DC_1ST_CLAMP2.Visu_Ret_Arr[13] := FALSE;
   S705_TL_DC_1ST_CLAMP2.Visu_Ret_Arr[14] := FALSE;
   S705_TL_DC_1ST_CLAMP2.Visu_Ret_Arr[15] := FALSE;
   S705_TL_DC_1ST_CLAMP2.BLK_Move_Ret := 0;
   S705_TL_DC_1ST_CLAMP2.Enable := TRUE;
   S705_TL_DC_1ST_CLAMP2.Adv_End := FALSE;
   S705_TL_DC_1ST_CLAMP2.Ret_End := TRUE;
   S705_TL_DC_1ST_CLAMP3.Enable_Aux := TRUE;
   S705_TL_DC_1ST_CLAMP3.Adv_Amount := 1;
   S705_TL_DC_1ST_CLAMP3.Ret_Amount := 3;
   S705_TL_DC_1ST_CLAMP3.LS_Adv1 := FALSE;
   S705_TL_DC_1ST_CLAMP3.LS_Ret1 := TRUE;
   S705_TL_DC_1ST_CLAMP3.LS_Adv2 := FALSE;
   S705_TL_DC_1ST_CLAMP3.LS_Ret2 := TRUE;
   S705_TL_DC_1ST_CLAMP3.LS_Adv3 := FALSE;
   S705_TL_DC_1ST_CLAMP3.LS_Ret3 := TRUE;
   S705_TL_DC_1ST_CLAMP3.LS_Adv4 := FALSE;
   S705_TL_DC_1ST_CLAMP3.LS_Ret4 := FALSE;
   S705_TL_DC_1ST_CLAMP3.LS_Adv5 := FALSE;
   S705_TL_DC_1ST_CLAMP3.LS_Ret5 := FALSE;
   S705_TL_DC_1ST_CLAMP3.LS_Adv6 := FALSE;
   S705_TL_DC_1ST_CLAMP3.LS_Ret6 := FALSE;
   S705_TL_DC_1ST_CLAMP3.LS_Adv7 := FALSE;
   S705_TL_DC_1ST_CLAMP3.LS_Ret7 := FALSE;
   S705_TL_DC_1ST_CLAMP3.LS_Adv8 := FALSE;
   S705_TL_DC_1ST_CLAMP3.LS_Ret8 := FALSE;
   S705_TL_DC_1ST_CLAMP3.SOL_Adv := FALSE;
   S705_TL_DC_1ST_CLAMP3.SOL_Ret := FALSE;
   S705_TL_DC_1ST_CLAMP3.M_Ready := TRUE;
   S705_TL_DC_1ST_CLAMP3.T_CHK1 := T#4S;
   S705_TL_DC_1ST_CLAMP3.T_CHK2 := T#4S;
   S705_TL_DC_1ST_CLAMP3.PB_Lamp_CHK := FALSE;
   S705_TL_DC_1ST_CLAMP3.PB_Error_Rst := FALSE;
   S705_TL_DC_1ST_CLAMP3.M_FLICK := TRUE;
   S705_TL_DC_1ST_CLAMP3.M_Adv_Err := FALSE;
   S705_TL_DC_1ST_CLAMP3.M_Ret_Err := FALSE;
   S705_TL_DC_1ST_CLAMP3.LP_Adv := FALSE;
   S705_TL_DC_1ST_CLAMP3.LP_Ret := TRUE;
   S705_TL_DC_1ST_CLAMP3.Visu_Adv := W#16#0;
   S705_TL_DC_1ST_CLAMP3.Visu_Ret := W#16#F00;
   S705_TL_DC_1ST_CLAMP3.Error_T1.IN := FALSE;
   S705_TL_DC_1ST_CLAMP3.Error_T1.PT := T#4S;
   S705_TL_DC_1ST_CLAMP3.Error_T1.Q := FALSE;
   S705_TL_DC_1ST_CLAMP3.Error_T1.ET := T#0MS;
   S705_TL_DC_1ST_CLAMP3.Error_T1.STATE := B#16#0;
   S705_TL_DC_1ST_CLAMP3.Error_T1.STIME := T#23D5H8M48S572MS;
   S705_TL_DC_1ST_CLAMP3.Error_T1.ATIME := T#23D5H8M50S65MS;
   S705_TL_DC_1ST_CLAMP3.Error_T2.IN := FALSE;
   S705_TL_DC_1ST_CLAMP3.Error_T2.PT := T#4S;
   S705_TL_DC_1ST_CLAMP3.Error_T2.Q := FALSE;
   S705_TL_DC_1ST_CLAMP3.Error_T2.ET := T#0MS;
   S705_TL_DC_1ST_CLAMP3.Error_T2.STATE := B#16#0;
   S705_TL_DC_1ST_CLAMP3.Error_T2.STIME := T#0MS;
   S705_TL_DC_1ST_CLAMP3.Error_T2.ATIME := T#0MS;
   S705_TL_DC_1ST_CLAMP3.Adv_End_Aux := FALSE;
   S705_TL_DC_1ST_CLAMP3.Ret_End_Aux := TRUE;
   S705_TL_DC_1ST_CLAMP3.CHK_Aux1 := FALSE;
   S705_TL_DC_1ST_CLAMP3.CHK_Aux2 := FALSE;
   S705_TL_DC_1ST_CLAMP3.Error_T1_DN := FALSE;
   S705_TL_DC_1ST_CLAMP3.Error_T2_DN := FALSE;
   S705_TL_DC_1ST_CLAMP3.Adv_Memo := FALSE;
   S705_TL_DC_1ST_CLAMP3.Visu_Adv_Arr[0] := FALSE;
   S705_TL_DC_1ST_CLAMP3.Visu_Adv_Arr[1] := FALSE;
   S705_TL_DC_1ST_CLAMP3.Visu_Adv_Arr[2] := FALSE;
   S705_TL_DC_1ST_CLAMP3.Visu_Adv_Arr[3] := FALSE;
   S705_TL_DC_1ST_CLAMP3.Visu_Adv_Arr[4] := FALSE;
   S705_TL_DC_1ST_CLAMP3.Visu_Adv_Arr[5] := FALSE;
   S705_TL_DC_1ST_CLAMP3.Visu_Adv_Arr[6] := FALSE;
   S705_TL_DC_1ST_CLAMP3.Visu_Adv_Arr[7] := FALSE;
   S705_TL_DC_1ST_CLAMP3.Visu_Adv_Arr[8] := FALSE;
   S705_TL_DC_1ST_CLAMP3.Visu_Adv_Arr[9] := FALSE;
   S705_TL_DC_1ST_CLAMP3.Visu_Adv_Arr[10] := FALSE;
   S705_TL_DC_1ST_CLAMP3.Visu_Adv_Arr[11] := FALSE;
   S705_TL_DC_1ST_CLAMP3.Visu_Adv_Arr[12] := FALSE;
   S705_TL_DC_1ST_CLAMP3.Visu_Adv_Arr[13] := FALSE;
   S705_TL_DC_1ST_CLAMP3.Visu_Adv_Arr[14] := FALSE;
   S705_TL_DC_1ST_CLAMP3.Visu_Adv_Arr[15] := FALSE;
   S705_TL_DC_1ST_CLAMP3.Visu_Ret_Arr[0] := TRUE;
   S705_TL_DC_1ST_CLAMP3.Visu_Ret_Arr[1] := TRUE;
   S705_TL_DC_1ST_CLAMP3.Visu_Ret_Arr[2] := TRUE;
   S705_TL_DC_1ST_CLAMP3.Visu_Ret_Arr[3] := TRUE;
   S705_TL_DC_1ST_CLAMP3.Visu_Ret_Arr[4] := FALSE;
   S705_TL_DC_1ST_CLAMP3.Visu_Ret_Arr[5] := FALSE;
   S705_TL_DC_1ST_CLAMP3.Visu_Ret_Arr[6] := FALSE;
   S705_TL_DC_1ST_CLAMP3.Visu_Ret_Arr[7] := FALSE;
   S705_TL_DC_1ST_CLAMP3.Visu_Ret_Arr[8] := FALSE;
   S705_TL_DC_1ST_CLAMP3.Visu_Ret_Arr[9] := FALSE;
   S705_TL_DC_1ST_CLAMP3.Visu_Ret_Arr[10] := FALSE;
   S705_TL_DC_1ST_CLAMP3.Visu_Ret_Arr[11] := FALSE;
   S705_TL_DC_1ST_CLAMP3.Visu_Ret_Arr[12] := FALSE;
   S705_TL_DC_1ST_CLAMP3.Visu_Ret_Arr[13] := FALSE;
   S705_TL_DC_1ST_CLAMP3.Visu_Ret_Arr[14] := FALSE;
   S705_TL_DC_1ST_CLAMP3.Visu_Ret_Arr[15] := FALSE;
   S705_TL_DC_1ST_CLAMP3.BLK_Move_Ret := 0;
   S705_TL_DC_1ST_CLAMP3.Enable := TRUE;
   S705_TL_DC_1ST_CLAMP3.Adv_End := FALSE;
   S705_TL_DC_1ST_CLAMP3.Ret_End := TRUE;
   S705_TL_DC_2ND_CLAMP1.Enable_Aux := TRUE;
   S705_TL_DC_2ND_CLAMP1.Adv_Amount := 1;
   S705_TL_DC_2ND_CLAMP1.Ret_Amount := 5;
   S705_TL_DC_2ND_CLAMP1.LS_Adv1 := FALSE;
   S705_TL_DC_2ND_CLAMP1.LS_Ret1 := TRUE;
   S705_TL_DC_2ND_CLAMP1.LS_Adv2 := FALSE;
   S705_TL_DC_2ND_CLAMP1.LS_Ret2 := TRUE;
   S705_TL_DC_2ND_CLAMP1.LS_Adv3 := FALSE;
   S705_TL_DC_2ND_CLAMP1.LS_Ret3 := TRUE;
   S705_TL_DC_2ND_CLAMP1.LS_Adv4 := FALSE;
   S705_TL_DC_2ND_CLAMP1.LS_Ret4 := TRUE;
   S705_TL_DC_2ND_CLAMP1.LS_Adv5 := FALSE;
   S705_TL_DC_2ND_CLAMP1.LS_Ret5 := TRUE;
   S705_TL_DC_2ND_CLAMP1.LS_Adv6 := FALSE;
   S705_TL_DC_2ND_CLAMP1.LS_Ret6 := FALSE;
   S705_TL_DC_2ND_CLAMP1.LS_Adv7 := FALSE;
   S705_TL_DC_2ND_CLAMP1.LS_Ret7 := FALSE;
   S705_TL_DC_2ND_CLAMP1.LS_Adv8 := FALSE;
   S705_TL_DC_2ND_CLAMP1.LS_Ret8 := FALSE;
   S705_TL_DC_2ND_CLAMP1.SOL_Adv := FALSE;
   S705_TL_DC_2ND_CLAMP1.SOL_Ret := FALSE;
   S705_TL_DC_2ND_CLAMP1.M_Ready := TRUE;
   S705_TL_DC_2ND_CLAMP1.T_CHK1 := T#4S;
   S705_TL_DC_2ND_CLAMP1.T_CHK2 := T#4S;
   S705_TL_DC_2ND_CLAMP1.PB_Lamp_CHK := FALSE;
   S705_TL_DC_2ND_CLAMP1.PB_Error_Rst := FALSE;
   S705_TL_DC_2ND_CLAMP1.M_FLICK := TRUE;
   S705_TL_DC_2ND_CLAMP1.M_Adv_Err := FALSE;
   S705_TL_DC_2ND_CLAMP1.M_Ret_Err := FALSE;
   S705_TL_DC_2ND_CLAMP1.LP_Adv := FALSE;
   S705_TL_DC_2ND_CLAMP1.LP_Ret := TRUE;
   S705_TL_DC_2ND_CLAMP1.Visu_Adv := W#16#0;
   S705_TL_DC_2ND_CLAMP1.Visu_Ret := W#16#3F00;
   S705_TL_DC_2ND_CLAMP1.Error_T1.IN := FALSE;
   S705_TL_DC_2ND_CLAMP1.Error_T1.PT := T#4S;
   S705_TL_DC_2ND_CLAMP1.Error_T1.Q := FALSE;
   S705_TL_DC_2ND_CLAMP1.Error_T1.ET := T#0MS;
   S705_TL_DC_2ND_CLAMP1.Error_T1.STATE := B#16#0;
   S705_TL_DC_2ND_CLAMP1.Error_T1.STIME := T#23D5H8M48S572MS;
   S705_TL_DC_2ND_CLAMP1.Error_T1.ATIME := T#23D5H8M49S880MS;
   S705_TL_DC_2ND_CLAMP1.Error_T2.IN := FALSE;
   S705_TL_DC_2ND_CLAMP1.Error_T2.PT := T#4S;
   S705_TL_DC_2ND_CLAMP1.Error_T2.Q := FALSE;
   S705_TL_DC_2ND_CLAMP1.Error_T2.ET := T#0MS;
   S705_TL_DC_2ND_CLAMP1.Error_T2.STATE := B#16#0;
   S705_TL_DC_2ND_CLAMP1.Error_T2.STIME := T#0MS;
   S705_TL_DC_2ND_CLAMP1.Error_T2.ATIME := T#0MS;
   S705_TL_DC_2ND_CLAMP1.Adv_End_Aux := FALSE;
   S705_TL_DC_2ND_CLAMP1.Ret_End_Aux := TRUE;
   S705_TL_DC_2ND_CLAMP1.CHK_Aux1 := FALSE;
   S705_TL_DC_2ND_CLAMP1.CHK_Aux2 := FALSE;
   S705_TL_DC_2ND_CLAMP1.Error_T1_DN := FALSE;
   S705_TL_DC_2ND_CLAMP1.Error_T2_DN := FALSE;
   S705_TL_DC_2ND_CLAMP1.Adv_Memo := FALSE;
   S705_TL_DC_2ND_CLAMP1.Visu_Adv_Arr[0] := FALSE;
   S705_TL_DC_2ND_CLAMP1.Visu_Adv_Arr[1] := FALSE;
   S705_TL_DC_2ND_CLAMP1.Visu_Adv_Arr[2] := FALSE;
   S705_TL_DC_2ND_CLAMP1.Visu_Adv_Arr[3] := FALSE;
   S705_TL_DC_2ND_CLAMP1.Visu_Adv_Arr[4] := FALSE;
   S705_TL_DC_2ND_CLAMP1.Visu_Adv_Arr[5] := FALSE;
   S705_TL_DC_2ND_CLAMP1.Visu_Adv_Arr[6] := FALSE;
   S705_TL_DC_2ND_CLAMP1.Visu_Adv_Arr[7] := FALSE;
   S705_TL_DC_2ND_CLAMP1.Visu_Adv_Arr[8] := FALSE;
   S705_TL_DC_2ND_CLAMP1.Visu_Adv_Arr[9] := FALSE;
   S705_TL_DC_2ND_CLAMP1.Visu_Adv_Arr[10] := FALSE;
   S705_TL_DC_2ND_CLAMP1.Visu_Adv_Arr[11] := FALSE;
   S705_TL_DC_2ND_CLAMP1.Visu_Adv_Arr[12] := FALSE;
   S705_TL_DC_2ND_CLAMP1.Visu_Adv_Arr[13] := FALSE;
   S705_TL_DC_2ND_CLAMP1.Visu_Adv_Arr[14] := FALSE;
   S705_TL_DC_2ND_CLAMP1.Visu_Adv_Arr[15] := FALSE;
   S705_TL_DC_2ND_CLAMP1.Visu_Ret_Arr[0] := TRUE;
   S705_TL_DC_2ND_CLAMP1.Visu_Ret_Arr[1] := TRUE;
   S705_TL_DC_2ND_CLAMP1.Visu_Ret_Arr[2] := TRUE;
   S705_TL_DC_2ND_CLAMP1.Visu_Ret_Arr[3] := TRUE;
   S705_TL_DC_2ND_CLAMP1.Visu_Ret_Arr[4] := TRUE;
   S705_TL_DC_2ND_CLAMP1.Visu_Ret_Arr[5] := TRUE;
   S705_TL_DC_2ND_CLAMP1.Visu_Ret_Arr[6] := FALSE;
   S705_TL_DC_2ND_CLAMP1.Visu_Ret_Arr[7] := FALSE;
   S705_TL_DC_2ND_CLAMP1.Visu_Ret_Arr[8] := FALSE;
   S705_TL_DC_2ND_CLAMP1.Visu_Ret_Arr[9] := FALSE;
   S705_TL_DC_2ND_CLAMP1.Visu_Ret_Arr[10] := FALSE;
   S705_TL_DC_2ND_CLAMP1.Visu_Ret_Arr[11] := FALSE;
   S705_TL_DC_2ND_CLAMP1.Visu_Ret_Arr[12] := FALSE;
   S705_TL_DC_2ND_CLAMP1.Visu_Ret_Arr[13] := FALSE;
   S705_TL_DC_2ND_CLAMP1.Visu_Ret_Arr[14] := FALSE;
   S705_TL_DC_2ND_CLAMP1.Visu_Ret_Arr[15] := FALSE;
   S705_TL_DC_2ND_CLAMP1.BLK_Move_Ret := 0;
   S705_TL_DC_2ND_CLAMP1.Enable := TRUE;
   S705_TL_DC_2ND_CLAMP1.Adv_End := FALSE;
   S705_TL_DC_2ND_CLAMP1.Ret_End := TRUE;
   S705_TL_DC_2ND_CLAMP2.Enable_Aux := TRUE;
   S705_TL_DC_2ND_CLAMP2.Adv_Amount := 1;
   S705_TL_DC_2ND_CLAMP2.Ret_Amount := 5;
   S705_TL_DC_2ND_CLAMP2.LS_Adv1 := FALSE;
   S705_TL_DC_2ND_CLAMP2.LS_Ret1 := TRUE;
   S705_TL_DC_2ND_CLAMP2.LS_Adv2 := FALSE;
   S705_TL_DC_2ND_CLAMP2.LS_Ret2 := TRUE;
   S705_TL_DC_2ND_CLAMP2.LS_Adv3 := FALSE;
   S705_TL_DC_2ND_CLAMP2.LS_Ret3 := TRUE;
   S705_TL_DC_2ND_CLAMP2.LS_Adv4 := FALSE;
   S705_TL_DC_2ND_CLAMP2.LS_Ret4 := TRUE;
   S705_TL_DC_2ND_CLAMP2.LS_Adv5 := FALSE;
   S705_TL_DC_2ND_CLAMP2.LS_Ret5 := TRUE;
   S705_TL_DC_2ND_CLAMP2.LS_Adv6 := FALSE;
   S705_TL_DC_2ND_CLAMP2.LS_Ret6 := FALSE;
   S705_TL_DC_2ND_CLAMP2.LS_Adv7 := FALSE;
   S705_TL_DC_2ND_CLAMP2.LS_Ret7 := FALSE;
   S705_TL_DC_2ND_CLAMP2.LS_Adv8 := FALSE;
   S705_TL_DC_2ND_CLAMP2.LS_Ret8 := FALSE;
   S705_TL_DC_2ND_CLAMP2.SOL_Adv := FALSE;
   S705_TL_DC_2ND_CLAMP2.SOL_Ret := FALSE;
   S705_TL_DC_2ND_CLAMP2.M_Ready := TRUE;
   S705_TL_DC_2ND_CLAMP2.T_CHK1 := T#4S;
   S705_TL_DC_2ND_CLAMP2.T_CHK2 := T#4S;
   S705_TL_DC_2ND_CLAMP2.PB_Lamp_CHK := FALSE;
   S705_TL_DC_2ND_CLAMP2.PB_Error_Rst := FALSE;
   S705_TL_DC_2ND_CLAMP2.M_FLICK := TRUE;
   S705_TL_DC_2ND_CLAMP2.M_Adv_Err := FALSE;
   S705_TL_DC_2ND_CLAMP2.M_Ret_Err := FALSE;
   S705_TL_DC_2ND_CLAMP2.LP_Adv := FALSE;
   S705_TL_DC_2ND_CLAMP2.LP_Ret := TRUE;
   S705_TL_DC_2ND_CLAMP2.Visu_Adv := W#16#0;
   S705_TL_DC_2ND_CLAMP2.Visu_Ret := W#16#3F00;
   S705_TL_DC_2ND_CLAMP2.Error_T1.IN := FALSE;
   S705_TL_DC_2ND_CLAMP2.Error_T1.PT := T#4S;
   S705_TL_DC_2ND_CLAMP2.Error_T1.Q := FALSE;
   S705_TL_DC_2ND_CLAMP2.Error_T1.ET := T#0MS;
   S705_TL_DC_2ND_CLAMP2.Error_T1.STATE := B#16#0;
   S705_TL_DC_2ND_CLAMP2.Error_T1.STIME := T#23D5H8M48S572MS;
   S705_TL_DC_2ND_CLAMP2.Error_T1.ATIME := T#23D5H8M50S18MS;
   S705_TL_DC_2ND_CLAMP2.Error_T2.IN := FALSE;
   S705_TL_DC_2ND_CLAMP2.Error_T2.PT := T#4S;
   S705_TL_DC_2ND_CLAMP2.Error_T2.Q := FALSE;
   S705_TL_DC_2ND_CLAMP2.Error_T2.ET := T#0MS;
   S705_TL_DC_2ND_CLAMP2.Error_T2.STATE := B#16#0;
   S705_TL_DC_2ND_CLAMP2.Error_T2.STIME := T#0MS;
   S705_TL_DC_2ND_CLAMP2.Error_T2.ATIME := T#0MS;
   S705_TL_DC_2ND_CLAMP2.Adv_End_Aux := FALSE;
   S705_TL_DC_2ND_CLAMP2.Ret_End_Aux := TRUE;
   S705_TL_DC_2ND_CLAMP2.CHK_Aux1 := FALSE;
   S705_TL_DC_2ND_CLAMP2.CHK_Aux2 := FALSE;
   S705_TL_DC_2ND_CLAMP2.Error_T1_DN := FALSE;
   S705_TL_DC_2ND_CLAMP2.Error_T2_DN := FALSE;
   S705_TL_DC_2ND_CLAMP2.Adv_Memo := FALSE;
   S705_TL_DC_2ND_CLAMP2.Visu_Adv_Arr[0] := FALSE;
   S705_TL_DC_2ND_CLAMP2.Visu_Adv_Arr[1] := FALSE;
   S705_TL_DC_2ND_CLAMP2.Visu_Adv_Arr[2] := FALSE;
   S705_TL_DC_2ND_CLAMP2.Visu_Adv_Arr[3] := FALSE;
   S705_TL_DC_2ND_CLAMP2.Visu_Adv_Arr[4] := FALSE;
   S705_TL_DC_2ND_CLAMP2.Visu_Adv_Arr[5] := FALSE;
   S705_TL_DC_2ND_CLAMP2.Visu_Adv_Arr[6] := FALSE;
   S705_TL_DC_2ND_CLAMP2.Visu_Adv_Arr[7] := FALSE;
   S705_TL_DC_2ND_CLAMP2.Visu_Adv_Arr[8] := FALSE;
   S705_TL_DC_2ND_CLAMP2.Visu_Adv_Arr[9] := FALSE;
   S705_TL_DC_2ND_CLAMP2.Visu_Adv_Arr[10] := FALSE;
   S705_TL_DC_2ND_CLAMP2.Visu_Adv_Arr[11] := FALSE;
   S705_TL_DC_2ND_CLAMP2.Visu_Adv_Arr[12] := FALSE;
   S705_TL_DC_2ND_CLAMP2.Visu_Adv_Arr[13] := FALSE;
   S705_TL_DC_2ND_CLAMP2.Visu_Adv_Arr[14] := FALSE;
   S705_TL_DC_2ND_CLAMP2.Visu_Adv_Arr[15] := FALSE;
   S705_TL_DC_2ND_CLAMP2.Visu_Ret_Arr[0] := TRUE;
   S705_TL_DC_2ND_CLAMP2.Visu_Ret_Arr[1] := TRUE;
   S705_TL_DC_2ND_CLAMP2.Visu_Ret_Arr[2] := TRUE;
   S705_TL_DC_2ND_CLAMP2.Visu_Ret_Arr[3] := TRUE;
   S705_TL_DC_2ND_CLAMP2.Visu_Ret_Arr[4] := TRUE;
   S705_TL_DC_2ND_CLAMP2.Visu_Ret_Arr[5] := TRUE;
   S705_TL_DC_2ND_CLAMP2.Visu_Ret_Arr[6] := FALSE;
   S705_TL_DC_2ND_CLAMP2.Visu_Ret_Arr[7] := FALSE;
   S705_TL_DC_2ND_CLAMP2.Visu_Ret_Arr[8] := FALSE;
   S705_TL_DC_2ND_CLAMP2.Visu_Ret_Arr[9] := FALSE;
   S705_TL_DC_2ND_CLAMP2.Visu_Ret_Arr[10] := FALSE;
   S705_TL_DC_2ND_CLAMP2.Visu_Ret_Arr[11] := FALSE;
   S705_TL_DC_2ND_CLAMP2.Visu_Ret_Arr[12] := FALSE;
   S705_TL_DC_2ND_CLAMP2.Visu_Ret_Arr[13] := FALSE;
   S705_TL_DC_2ND_CLAMP2.Visu_Ret_Arr[14] := FALSE;
   S705_TL_DC_2ND_CLAMP2.Visu_Ret_Arr[15] := FALSE;
   S705_TL_DC_2ND_CLAMP2.BLK_Move_Ret := 0;
   S705_TL_DC_2ND_CLAMP2.Enable := TRUE;
   S705_TL_DC_2ND_CLAMP2.Adv_End := FALSE;
   S705_TL_DC_2ND_CLAMP2.Ret_End := TRUE;
   S705_TL_DC_U261.Enable_Aux := TRUE;
   S705_TL_DC_U261.Adv_Amount := 1;
   S705_TL_DC_U261.Ret_Amount := 1;
   S705_TL_DC_U261.LS_Adv1 := FALSE;
   S705_TL_DC_U261.LS_Ret1 := TRUE;
   S705_TL_DC_U261.LS_Adv2 := FALSE;
   S705_TL_DC_U261.LS_Ret2 := FALSE;
   S705_TL_DC_U261.LS_Adv3 := FALSE;
   S705_TL_DC_U261.LS_Ret3 := FALSE;
   S705_TL_DC_U261.LS_Adv4 := FALSE;
   S705_TL_DC_U261.LS_Ret4 := FALSE;
   S705_TL_DC_U261.LS_Adv5 := FALSE;
   S705_TL_DC_U261.LS_Ret5 := FALSE;
   S705_TL_DC_U261.LS_Adv6 := FALSE;
   S705_TL_DC_U261.LS_Ret6 := FALSE;
   S705_TL_DC_U261.LS_Adv7 := FALSE;
   S705_TL_DC_U261.LS_Ret7 := FALSE;
   S705_TL_DC_U261.LS_Adv8 := FALSE;
   S705_TL_DC_U261.LS_Ret8 := FALSE;
   S705_TL_DC_U261.SOL_Adv := FALSE;
   S705_TL_DC_U261.SOL_Ret := FALSE;
   S705_TL_DC_U261.M_Ready := TRUE;
   S705_TL_DC_U261.T_CHK1 := T#4S;
   S705_TL_DC_U261.T_CHK2 := T#4S;
   S705_TL_DC_U261.PB_Lamp_CHK := FALSE;
   S705_TL_DC_U261.PB_Error_Rst := FALSE;
   S705_TL_DC_U261.M_FLICK := TRUE;
   S705_TL_DC_U261.M_Adv_Err := FALSE;
   S705_TL_DC_U261.M_Ret_Err := FALSE;
   S705_TL_DC_U261.LP_Adv := FALSE;
   S705_TL_DC_U261.LP_Ret := TRUE;
   S705_TL_DC_U261.Visu_Adv := W#16#0;
   S705_TL_DC_U261.Visu_Ret := W#16#100;
   S705_TL_DC_U261.Error_T1.IN := FALSE;
   S705_TL_DC_U261.Error_T1.PT := T#4S;
   S705_TL_DC_U261.Error_T1.Q := FALSE;
   S705_TL_DC_U261.Error_T1.ET := T#0MS;
   S705_TL_DC_U261.Error_T1.STATE := B#16#0;
   S705_TL_DC_U261.Error_T1.STIME := T#23D5H8M46S915MS;
   S705_TL_DC_U261.Error_T1.ATIME := T#23D5H8M46S961MS;
   S705_TL_DC_U261.Error_T2.IN := FALSE;
   S705_TL_DC_U261.Error_T2.PT := T#4S;
   S705_TL_DC_U261.Error_T2.Q := FALSE;
   S705_TL_DC_U261.Error_T2.ET := T#0MS;
   S705_TL_DC_U261.Error_T2.STATE := B#16#0;
   S705_TL_DC_U261.Error_T2.STIME := T#0MS;
   S705_TL_DC_U261.Error_T2.ATIME := T#0MS;
   S705_TL_DC_U261.Adv_End_Aux := FALSE;
   S705_TL_DC_U261.Ret_End_Aux := TRUE;
   S705_TL_DC_U261.CHK_Aux1 := FALSE;
   S705_TL_DC_U261.CHK_Aux2 := FALSE;
   S705_TL_DC_U261.Error_T1_DN := FALSE;
   S705_TL_DC_U261.Error_T2_DN := FALSE;
   S705_TL_DC_U261.Adv_Memo := TRUE;
   S705_TL_DC_U261.Visu_Adv_Arr[0] := FALSE;
   S705_TL_DC_U261.Visu_Adv_Arr[1] := FALSE;
   S705_TL_DC_U261.Visu_Adv_Arr[2] := FALSE;
   S705_TL_DC_U261.Visu_Adv_Arr[3] := FALSE;
   S705_TL_DC_U261.Visu_Adv_Arr[4] := FALSE;
   S705_TL_DC_U261.Visu_Adv_Arr[5] := FALSE;
   S705_TL_DC_U261.Visu_Adv_Arr[6] := FALSE;
   S705_TL_DC_U261.Visu_Adv_Arr[7] := FALSE;
   S705_TL_DC_U261.Visu_Adv_Arr[8] := FALSE;
   S705_TL_DC_U261.Visu_Adv_Arr[9] := FALSE;
   S705_TL_DC_U261.Visu_Adv_Arr[10] := FALSE;
   S705_TL_DC_U261.Visu_Adv_Arr[11] := FALSE;
   S705_TL_DC_U261.Visu_Adv_Arr[12] := FALSE;
   S705_TL_DC_U261.Visu_Adv_Arr[13] := FALSE;
   S705_TL_DC_U261.Visu_Adv_Arr[14] := FALSE;
   S705_TL_DC_U261.Visu_Adv_Arr[15] := FALSE;
   S705_TL_DC_U261.Visu_Ret_Arr[0] := TRUE;
   S705_TL_DC_U261.Visu_Ret_Arr[1] := FALSE;
   S705_TL_DC_U261.Visu_Ret_Arr[2] := FALSE;
   S705_TL_DC_U261.Visu_Ret_Arr[3] := FALSE;
   S705_TL_DC_U261.Visu_Ret_Arr[4] := FALSE;
   S705_TL_DC_U261.Visu_Ret_Arr[5] := FALSE;
   S705_TL_DC_U261.Visu_Ret_Arr[6] := FALSE;
   S705_TL_DC_U261.Visu_Ret_Arr[7] := FALSE;
   S705_TL_DC_U261.Visu_Ret_Arr[8] := FALSE;
   S705_TL_DC_U261.Visu_Ret_Arr[9] := FALSE;
   S705_TL_DC_U261.Visu_Ret_Arr[10] := FALSE;
   S705_TL_DC_U261.Visu_Ret_Arr[11] := FALSE;
   S705_TL_DC_U261.Visu_Ret_Arr[12] := FALSE;
   S705_TL_DC_U261.Visu_Ret_Arr[13] := FALSE;
   S705_TL_DC_U261.Visu_Ret_Arr[14] := FALSE;
   S705_TL_DC_U261.Visu_Ret_Arr[15] := FALSE;
   S705_TL_DC_U261.BLK_Move_Ret := 0;
   S705_TL_DC_U261.Enable := TRUE;
   S705_TL_DC_U261.Adv_End := FALSE;
   S705_TL_DC_U261.Ret_End := TRUE;
   S705_TL_DC_U261_CLAMP.Enable_Aux := TRUE;
   S705_TL_DC_U261_CLAMP.Adv_Amount := 1;
   S705_TL_DC_U261_CLAMP.Ret_Amount := 1;
   S705_TL_DC_U261_CLAMP.LS_Adv1 := FALSE;
   S705_TL_DC_U261_CLAMP.LS_Ret1 := TRUE;
   S705_TL_DC_U261_CLAMP.LS_Adv2 := FALSE;
   S705_TL_DC_U261_CLAMP.LS_Ret2 := FALSE;
   S705_TL_DC_U261_CLAMP.LS_Adv3 := FALSE;
   S705_TL_DC_U261_CLAMP.LS_Ret3 := FALSE;
   S705_TL_DC_U261_CLAMP.LS_Adv4 := FALSE;
   S705_TL_DC_U261_CLAMP.LS_Ret4 := FALSE;
   S705_TL_DC_U261_CLAMP.LS_Adv5 := FALSE;
   S705_TL_DC_U261_CLAMP.LS_Ret5 := FALSE;
   S705_TL_DC_U261_CLAMP.LS_Adv6 := FALSE;
   S705_TL_DC_U261_CLAMP.LS_Ret6 := FALSE;
   S705_TL_DC_U261_CLAMP.LS_Adv7 := FALSE;
   S705_TL_DC_U261_CLAMP.LS_Ret7 := FALSE;
   S705_TL_DC_U261_CLAMP.LS_Adv8 := FALSE;
   S705_TL_DC_U261_CLAMP.LS_Ret8 := FALSE;
   S705_TL_DC_U261_CLAMP.SOL_Adv := FALSE;
   S705_TL_DC_U261_CLAMP.SOL_Ret := FALSE;
   S705_TL_DC_U261_CLAMP.M_Ready := TRUE;
   S705_TL_DC_U261_CLAMP.T_CHK1 := T#7S;
   S705_TL_DC_U261_CLAMP.T_CHK2 := T#7S;
   S705_TL_DC_U261_CLAMP.PB_Lamp_CHK := FALSE;
   S705_TL_DC_U261_CLAMP.PB_Error_Rst := FALSE;
   S705_TL_DC_U261_CLAMP.M_FLICK := TRUE;
   S705_TL_DC_U261_CLAMP.M_Adv_Err := FALSE;
   S705_TL_DC_U261_CLAMP.M_Ret_Err := FALSE;
   S705_TL_DC_U261_CLAMP.LP_Adv := FALSE;
   S705_TL_DC_U261_CLAMP.LP_Ret := TRUE;
   S705_TL_DC_U261_CLAMP.Visu_Adv := W#16#0;
   S705_TL_DC_U261_CLAMP.Visu_Ret := W#16#100;
   S705_TL_DC_U261_CLAMP.Error_T1.IN := FALSE;
   S705_TL_DC_U261_CLAMP.Error_T1.PT := T#7S;
   S705_TL_DC_U261_CLAMP.Error_T1.Q := FALSE;
   S705_TL_DC_U261_CLAMP.Error_T1.ET := T#0MS;
   S705_TL_DC_U261_CLAMP.Error_T1.STATE := B#16#0;
   S705_TL_DC_U261_CLAMP.Error_T1.STIME := T#23D5H8M46S916MS;
   S705_TL_DC_U261_CLAMP.Error_T1.ATIME := T#23D5H8M46S961MS;
   S705_TL_DC_U261_CLAMP.Error_T2.IN := FALSE;
   S705_TL_DC_U261_CLAMP.Error_T2.PT := T#7S;
   S705_TL_DC_U261_CLAMP.Error_T2.Q := FALSE;
   S705_TL_DC_U261_CLAMP.Error_T2.ET := T#0MS;
   S705_TL_DC_U261_CLAMP.Error_T2.STATE := B#16#0;
   S705_TL_DC_U261_CLAMP.Error_T2.STIME := T#0MS;
   S705_TL_DC_U261_CLAMP.Error_T2.ATIME := T#0MS;
   S705_TL_DC_U261_CLAMP.Adv_End_Aux := FALSE;
   S705_TL_DC_U261_CLAMP.Ret_End_Aux := TRUE;
   S705_TL_DC_U261_CLAMP.CHK_Aux1 := FALSE;
   S705_TL_DC_U261_CLAMP.CHK_Aux2 := FALSE;
   S705_TL_DC_U261_CLAMP.Error_T1_DN := FALSE;
   S705_TL_DC_U261_CLAMP.Error_T2_DN := FALSE;
   S705_TL_DC_U261_CLAMP.Adv_Memo := TRUE;
   S705_TL_DC_U261_CLAMP.Visu_Adv_Arr[0] := FALSE;
   S705_TL_DC_U261_CLAMP.Visu_Adv_Arr[1] := FALSE;
   S705_TL_DC_U261_CLAMP.Visu_Adv_Arr[2] := FALSE;
   S705_TL_DC_U261_CLAMP.Visu_Adv_Arr[3] := FALSE;
   S705_TL_DC_U261_CLAMP.Visu_Adv_Arr[4] := FALSE;
   S705_TL_DC_U261_CLAMP.Visu_Adv_Arr[5] := FALSE;
   S705_TL_DC_U261_CLAMP.Visu_Adv_Arr[6] := FALSE;
   S705_TL_DC_U261_CLAMP.Visu_Adv_Arr[7] := FALSE;
   S705_TL_DC_U261_CLAMP.Visu_Adv_Arr[8] := FALSE;
   S705_TL_DC_U261_CLAMP.Visu_Adv_Arr[9] := FALSE;
   S705_TL_DC_U261_CLAMP.Visu_Adv_Arr[10] := FALSE;
   S705_TL_DC_U261_CLAMP.Visu_Adv_Arr[11] := FALSE;
   S705_TL_DC_U261_CLAMP.Visu_Adv_Arr[12] := FALSE;
   S705_TL_DC_U261_CLAMP.Visu_Adv_Arr[13] := FALSE;
   S705_TL_DC_U261_CLAMP.Visu_Adv_Arr[14] := FALSE;
   S705_TL_DC_U261_CLAMP.Visu_Adv_Arr[15] := FALSE;
   S705_TL_DC_U261_CLAMP.Visu_Ret_Arr[0] := TRUE;
   S705_TL_DC_U261_CLAMP.Visu_Ret_Arr[1] := FALSE;
   S705_TL_DC_U261_CLAMP.Visu_Ret_Arr[2] := FALSE;
   S705_TL_DC_U261_CLAMP.Visu_Ret_Arr[3] := FALSE;
   S705_TL_DC_U261_CLAMP.Visu_Ret_Arr[4] := FALSE;
   S705_TL_DC_U261_CLAMP.Visu_Ret_Arr[5] := FALSE;
   S705_TL_DC_U261_CLAMP.Visu_Ret_Arr[6] := FALSE;
   S705_TL_DC_U261_CLAMP.Visu_Ret_Arr[7] := FALSE;
   S705_TL_DC_U261_CLAMP.Visu_Ret_Arr[8] := FALSE;
   S705_TL_DC_U261_CLAMP.Visu_Ret_Arr[9] := FALSE;
   S705_TL_DC_U261_CLAMP.Visu_Ret_Arr[10] := FALSE;
   S705_TL_DC_U261_CLAMP.Visu_Ret_Arr[11] := FALSE;
   S705_TL_DC_U261_CLAMP.Visu_Ret_Arr[12] := FALSE;
   S705_TL_DC_U261_CLAMP.Visu_Ret_Arr[13] := FALSE;
   S705_TL_DC_U261_CLAMP.Visu_Ret_Arr[14] := FALSE;
   S705_TL_DC_U261_CLAMP.Visu_Ret_Arr[15] := FALSE;
   S705_TL_DC_U261_CLAMP.BLK_Move_Ret := 0;
   S705_TL_DC_U261_CLAMP.Enable := TRUE;
   S705_TL_DC_U261_CLAMP.Adv_End := FALSE;
   S705_TL_DC_U261_CLAMP.Ret_End := TRUE;
   S705_TL_DC_U269.Enable_Aux := TRUE;
   S705_TL_DC_U269.Adv_Amount := 1;
   S705_TL_DC_U269.Ret_Amount := 1;
   S705_TL_DC_U269.LS_Adv1 := FALSE;
   S705_TL_DC_U269.LS_Ret1 := TRUE;
   S705_TL_DC_U269.LS_Adv2 := FALSE;
   S705_TL_DC_U269.LS_Ret2 := FALSE;
   S705_TL_DC_U269.LS_Adv3 := FALSE;
   S705_TL_DC_U269.LS_Ret3 := FALSE;
   S705_TL_DC_U269.LS_Adv4 := FALSE;
   S705_TL_DC_U269.LS_Ret4 := FALSE;
   S705_TL_DC_U269.LS_Adv5 := FALSE;
   S705_TL_DC_U269.LS_Ret5 := FALSE;
   S705_TL_DC_U269.LS_Adv6 := FALSE;
   S705_TL_DC_U269.LS_Ret6 := FALSE;
   S705_TL_DC_U269.LS_Adv7 := FALSE;
   S705_TL_DC_U269.LS_Ret7 := FALSE;
   S705_TL_DC_U269.LS_Adv8 := FALSE;
   S705_TL_DC_U269.LS_Ret8 := FALSE;
   S705_TL_DC_U269.SOL_Adv := FALSE;
   S705_TL_DC_U269.SOL_Ret := FALSE;
   S705_TL_DC_U269.M_Ready := TRUE;
   S705_TL_DC_U269.T_CHK1 := T#4S;
   S705_TL_DC_U269.T_CHK2 := T#4S;
   S705_TL_DC_U269.PB_Lamp_CHK := FALSE;
   S705_TL_DC_U269.PB_Error_Rst := FALSE;
   S705_TL_DC_U269.M_FLICK := TRUE;
   S705_TL_DC_U269.M_Adv_Err := FALSE;
   S705_TL_DC_U269.M_Ret_Err := FALSE;
   S705_TL_DC_U269.LP_Adv := FALSE;
   S705_TL_DC_U269.LP_Ret := TRUE;
   S705_TL_DC_U269.Visu_Adv := W#16#0;
   S705_TL_DC_U269.Visu_Ret := W#16#300;
   S705_TL_DC_U269.Error_T1.IN := FALSE;
   S705_TL_DC_U269.Error_T1.PT := T#4S;
   S705_TL_DC_U269.Error_T1.Q := FALSE;
   S705_TL_DC_U269.Error_T1.ET := T#0MS;
   S705_TL_DC_U269.Error_T1.STATE := B#16#0;
   S705_TL_DC_U269.Error_T1.STIME := T#23D5H8M49S9MS;
   S705_TL_DC_U269.Error_T1.ATIME := T#23D5H8M49S745MS;
   S705_TL_DC_U269.Error_T2.IN := FALSE;
   S705_TL_DC_U269.Error_T2.PT := T#4S;
   S705_TL_DC_U269.Error_T2.Q := FALSE;
   S705_TL_DC_U269.Error_T2.ET := T#0MS;
   S705_TL_DC_U269.Error_T2.STATE := B#16#0;
   S705_TL_DC_U269.Error_T2.STIME := T#0MS;
   S705_TL_DC_U269.Error_T2.ATIME := T#0MS;
   S705_TL_DC_U269.Adv_End_Aux := FALSE;
   S705_TL_DC_U269.Ret_End_Aux := TRUE;
   S705_TL_DC_U269.CHK_Aux1 := FALSE;
   S705_TL_DC_U269.CHK_Aux2 := FALSE;
   S705_TL_DC_U269.Error_T1_DN := FALSE;
   S705_TL_DC_U269.Error_T2_DN := FALSE;
   S705_TL_DC_U269.Adv_Memo := FALSE;
   S705_TL_DC_U269.Visu_Adv_Arr[0] := FALSE;
   S705_TL_DC_U269.Visu_Adv_Arr[1] := FALSE;
   S705_TL_DC_U269.Visu_Adv_Arr[2] := FALSE;
   S705_TL_DC_U269.Visu_Adv_Arr[3] := FALSE;
   S705_TL_DC_U269.Visu_Adv_Arr[4] := FALSE;
   S705_TL_DC_U269.Visu_Adv_Arr[5] := FALSE;
   S705_TL_DC_U269.Visu_Adv_Arr[6] := FALSE;
   S705_TL_DC_U269.Visu_Adv_Arr[7] := FALSE;
   S705_TL_DC_U269.Visu_Adv_Arr[8] := FALSE;
   S705_TL_DC_U269.Visu_Adv_Arr[9] := FALSE;
   S705_TL_DC_U269.Visu_Adv_Arr[10] := FALSE;
   S705_TL_DC_U269.Visu_Adv_Arr[11] := FALSE;
   S705_TL_DC_U269.Visu_Adv_Arr[12] := FALSE;
   S705_TL_DC_U269.Visu_Adv_Arr[13] := FALSE;
   S705_TL_DC_U269.Visu_Adv_Arr[14] := FALSE;
   S705_TL_DC_U269.Visu_Adv_Arr[15] := FALSE;
   S705_TL_DC_U269.Visu_Ret_Arr[0] := TRUE;
   S705_TL_DC_U269.Visu_Ret_Arr[1] := TRUE;
   S705_TL_DC_U269.Visu_Ret_Arr[2] := FALSE;
   S705_TL_DC_U269.Visu_Ret_Arr[3] := FALSE;
   S705_TL_DC_U269.Visu_Ret_Arr[4] := FALSE;
   S705_TL_DC_U269.Visu_Ret_Arr[5] := FALSE;
   S705_TL_DC_U269.Visu_Ret_Arr[6] := FALSE;
   S705_TL_DC_U269.Visu_Ret_Arr[7] := FALSE;
   S705_TL_DC_U269.Visu_Ret_Arr[8] := FALSE;
   S705_TL_DC_U269.Visu_Ret_Arr[9] := FALSE;
   S705_TL_DC_U269.Visu_Ret_Arr[10] := FALSE;
   S705_TL_DC_U269.Visu_Ret_Arr[11] := FALSE;
   S705_TL_DC_U269.Visu_Ret_Arr[12] := FALSE;
   S705_TL_DC_U269.Visu_Ret_Arr[13] := FALSE;
   S705_TL_DC_U269.Visu_Ret_Arr[14] := FALSE;
   S705_TL_DC_U269.Visu_Ret_Arr[15] := FALSE;
   S705_TL_DC_U269.BLK_Move_Ret := 0;
   S705_TL_DC_U269.Enable := TRUE;
   S705_TL_DC_U269.Adv_End := FALSE;
   S705_TL_DC_U269.Ret_End := TRUE;
   S705_TL_DC_U269_CLAMP.Enable_Aux := TRUE;
   S705_TL_DC_U269_CLAMP.Adv_Amount := 1;
   S705_TL_DC_U269_CLAMP.Ret_Amount := 2;
   S705_TL_DC_U269_CLAMP.LS_Adv1 := FALSE;
   S705_TL_DC_U269_CLAMP.LS_Ret1 := TRUE;
   S705_TL_DC_U269_CLAMP.LS_Adv2 := FALSE;
   S705_TL_DC_U269_CLAMP.LS_Ret2 := TRUE;
   S705_TL_DC_U269_CLAMP.LS_Adv3 := FALSE;
   S705_TL_DC_U269_CLAMP.LS_Ret3 := FALSE;
   S705_TL_DC_U269_CLAMP.LS_Adv4 := FALSE;
   S705_TL_DC_U269_CLAMP.LS_Ret4 := FALSE;
   S705_TL_DC_U269_CLAMP.LS_Adv5 := FALSE;
   S705_TL_DC_U269_CLAMP.LS_Ret5 := FALSE;
   S705_TL_DC_U269_CLAMP.LS_Adv6 := FALSE;
   S705_TL_DC_U269_CLAMP.LS_Ret6 := FALSE;
   S705_TL_DC_U269_CLAMP.LS_Adv7 := FALSE;
   S705_TL_DC_U269_CLAMP.LS_Ret7 := FALSE;
   S705_TL_DC_U269_CLAMP.LS_Adv8 := FALSE;
   S705_TL_DC_U269_CLAMP.LS_Ret8 := FALSE;
   S705_TL_DC_U269_CLAMP.SOL_Adv := FALSE;
   S705_TL_DC_U269_CLAMP.SOL_Ret := FALSE;
   S705_TL_DC_U269_CLAMP.M_Ready := TRUE;
   S705_TL_DC_U269_CLAMP.T_CHK1 := T#4S;
   S705_TL_DC_U269_CLAMP.T_CHK2 := T#4S;
   S705_TL_DC_U269_CLAMP.PB_Lamp_CHK := FALSE;
   S705_TL_DC_U269_CLAMP.PB_Error_Rst := FALSE;
   S705_TL_DC_U269_CLAMP.M_FLICK := TRUE;
   S705_TL_DC_U269_CLAMP.M_Adv_Err := FALSE;
   S705_TL_DC_U269_CLAMP.M_Ret_Err := FALSE;
   S705_TL_DC_U269_CLAMP.LP_Adv := FALSE;
   S705_TL_DC_U269_CLAMP.LP_Ret := TRUE;
   S705_TL_DC_U269_CLAMP.Visu_Adv := W#16#0;
   S705_TL_DC_U269_CLAMP.Visu_Ret := W#16#100;
   S705_TL_DC_U269_CLAMP.Error_T1.IN := FALSE;
   S705_TL_DC_U269_CLAMP.Error_T1.PT := T#4S;
   S705_TL_DC_U269_CLAMP.Error_T1.Q := FALSE;
   S705_TL_DC_U269_CLAMP.Error_T1.ET := T#0MS;
   S705_TL_DC_U269_CLAMP.Error_T1.STATE := B#16#0;
   S705_TL_DC_U269_CLAMP.Error_T1.STIME := T#23D5H8M46S916MS;
   S705_TL_DC_U269_CLAMP.Error_T1.ATIME := T#23D5H8M46S961MS;
   S705_TL_DC_U269_CLAMP.Error_T2.IN := FALSE;
   S705_TL_DC_U269_CLAMP.Error_T2.PT := T#4S;
   S705_TL_DC_U269_CLAMP.Error_T2.Q := FALSE;
   S705_TL_DC_U269_CLAMP.Error_T2.ET := T#0MS;
   S705_TL_DC_U269_CLAMP.Error_T2.STATE := B#16#0;
   S705_TL_DC_U269_CLAMP.Error_T2.STIME := T#0MS;
   S705_TL_DC_U269_CLAMP.Error_T2.ATIME := T#0MS;
   S705_TL_DC_U269_CLAMP.Adv_End_Aux := FALSE;
   S705_TL_DC_U269_CLAMP.Ret_End_Aux := TRUE;
   S705_TL_DC_U269_CLAMP.CHK_Aux1 := FALSE;
   S705_TL_DC_U269_CLAMP.CHK_Aux2 := FALSE;
   S705_TL_DC_U269_CLAMP.Error_T1_DN := FALSE;
   S705_TL_DC_U269_CLAMP.Error_T2_DN := FALSE;
   S705_TL_DC_U269_CLAMP.Adv_Memo := TRUE;
   S705_TL_DC_U269_CLAMP.Visu_Adv_Arr[0] := FALSE;
   S705_TL_DC_U269_CLAMP.Visu_Adv_Arr[1] := FALSE;
   S705_TL_DC_U269_CLAMP.Visu_Adv_Arr[2] := FALSE;
   S705_TL_DC_U269_CLAMP.Visu_Adv_Arr[3] := FALSE;
   S705_TL_DC_U269_CLAMP.Visu_Adv_Arr[4] := FALSE;
   S705_TL_DC_U269_CLAMP.Visu_Adv_Arr[5] := FALSE;
   S705_TL_DC_U269_CLAMP.Visu_Adv_Arr[6] := FALSE;
   S705_TL_DC_U269_CLAMP.Visu_Adv_Arr[7] := FALSE;
   S705_TL_DC_U269_CLAMP.Visu_Adv_Arr[8] := FALSE;
   S705_TL_DC_U269_CLAMP.Visu_Adv_Arr[9] := FALSE;
   S705_TL_DC_U269_CLAMP.Visu_Adv_Arr[10] := FALSE;
   S705_TL_DC_U269_CLAMP.Visu_Adv_Arr[11] := FALSE;
   S705_TL_DC_U269_CLAMP.Visu_Adv_Arr[12] := FALSE;
   S705_TL_DC_U269_CLAMP.Visu_Adv_Arr[13] := FALSE;
   S705_TL_DC_U269_CLAMP.Visu_Adv_Arr[14] := FALSE;
   S705_TL_DC_U269_CLAMP.Visu_Adv_Arr[15] := FALSE;
   S705_TL_DC_U269_CLAMP.Visu_Ret_Arr[0] := TRUE;
   S705_TL_DC_U269_CLAMP.Visu_Ret_Arr[1] := FALSE;
   S705_TL_DC_U269_CLAMP.Visu_Ret_Arr[2] := FALSE;
   S705_TL_DC_U269_CLAMP.Visu_Ret_Arr[3] := FALSE;
   S705_TL_DC_U269_CLAMP.Visu_Ret_Arr[4] := FALSE;
   S705_TL_DC_U269_CLAMP.Visu_Ret_Arr[5] := FALSE;
   S705_TL_DC_U269_CLAMP.Visu_Ret_Arr[6] := FALSE;
   S705_TL_DC_U269_CLAMP.Visu_Ret_Arr[7] := FALSE;
   S705_TL_DC_U269_CLAMP.Visu_Ret_Arr[8] := FALSE;
   S705_TL_DC_U269_CLAMP.Visu_Ret_Arr[9] := FALSE;
   S705_TL_DC_U269_CLAMP.Visu_Ret_Arr[10] := FALSE;
   S705_TL_DC_U269_CLAMP.Visu_Ret_Arr[11] := FALSE;
   S705_TL_DC_U269_CLAMP.Visu_Ret_Arr[12] := FALSE;
   S705_TL_DC_U269_CLAMP.Visu_Ret_Arr[13] := FALSE;
   S705_TL_DC_U269_CLAMP.Visu_Ret_Arr[14] := FALSE;
   S705_TL_DC_U269_CLAMP.Visu_Ret_Arr[15] := FALSE;
   S705_TL_DC_U269_CLAMP.BLK_Move_Ret := 0;
   S705_TL_DC_U269_CLAMP.Enable := TRUE;
   S705_TL_DC_U269_CLAMP.Adv_End := FALSE;
   S705_TL_DC_U269_CLAMP.Ret_End := TRUE;
   S705_TL_DC_3RD_CLAMP.Enable_Aux := TRUE;
   S705_TL_DC_3RD_CLAMP.Adv_Amount := 1;
   S705_TL_DC_3RD_CLAMP.Ret_Amount := 1;
   S705_TL_DC_3RD_CLAMP.LS_Adv1 := FALSE;
   S705_TL_DC_3RD_CLAMP.LS_Ret1 := TRUE;
   S705_TL_DC_3RD_CLAMP.LS_Adv2 := FALSE;
   S705_TL_DC_3RD_CLAMP.LS_Ret2 := FALSE;
   S705_TL_DC_3RD_CLAMP.LS_Adv3 := FALSE;
   S705_TL_DC_3RD_CLAMP.LS_Ret3 := FALSE;
   S705_TL_DC_3RD_CLAMP.LS_Adv4 := FALSE;
   S705_TL_DC_3RD_CLAMP.LS_Ret4 := FALSE;
   S705_TL_DC_3RD_CLAMP.LS_Adv5 := FALSE;
   S705_TL_DC_3RD_CLAMP.LS_Ret5 := FALSE;
   S705_TL_DC_3RD_CLAMP.LS_Adv6 := FALSE;
   S705_TL_DC_3RD_CLAMP.LS_Ret6 := FALSE;
   S705_TL_DC_3RD_CLAMP.LS_Adv7 := FALSE;
   S705_TL_DC_3RD_CLAMP.LS_Ret7 := FALSE;
   S705_TL_DC_3RD_CLAMP.LS_Adv8 := FALSE;
   S705_TL_DC_3RD_CLAMP.LS_Ret8 := FALSE;
   S705_TL_DC_3RD_CLAMP.SOL_Adv := FALSE;
   S705_TL_DC_3RD_CLAMP.SOL_Ret := FALSE;
   S705_TL_DC_3RD_CLAMP.M_Ready := TRUE;
   S705_TL_DC_3RD_CLAMP.T_CHK1 := T#4S;
   S705_TL_DC_3RD_CLAMP.T_CHK2 := T#4S;
   S705_TL_DC_3RD_CLAMP.PB_Lamp_CHK := FALSE;
   S705_TL_DC_3RD_CLAMP.PB_Error_Rst := FALSE;
   S705_TL_DC_3RD_CLAMP.M_FLICK := TRUE;
   S705_TL_DC_3RD_CLAMP.M_Adv_Err := FALSE;
   S705_TL_DC_3RD_CLAMP.M_Ret_Err := FALSE;
   S705_TL_DC_3RD_CLAMP.LP_Adv := FALSE;
   S705_TL_DC_3RD_CLAMP.LP_Ret := TRUE;
   S705_TL_DC_3RD_CLAMP.Visu_Adv := W#16#0;
   S705_TL_DC_3RD_CLAMP.Visu_Ret := W#16#300;
   S705_TL_DC_3RD_CLAMP.Error_T1.IN := FALSE;
   S705_TL_DC_3RD_CLAMP.Error_T1.PT := T#4S;
   S705_TL_DC_3RD_CLAMP.Error_T1.Q := FALSE;
   S705_TL_DC_3RD_CLAMP.Error_T1.ET := T#0MS;
   S705_TL_DC_3RD_CLAMP.Error_T1.STATE := B#16#0;
   S705_TL_DC_3RD_CLAMP.Error_T1.STIME := T#23D5H8M48S572MS;
   S705_TL_DC_3RD_CLAMP.Error_T1.ATIME := T#23D5H8M49S9MS;
   S705_TL_DC_3RD_CLAMP.Error_T2.IN := FALSE;
   S705_TL_DC_3RD_CLAMP.Error_T2.PT := T#4S;
   S705_TL_DC_3RD_CLAMP.Error_T2.Q := FALSE;
   S705_TL_DC_3RD_CLAMP.Error_T2.ET := T#0MS;
   S705_TL_DC_3RD_CLAMP.Error_T2.STATE := B#16#0;
   S705_TL_DC_3RD_CLAMP.Error_T2.STIME := T#0MS;
   S705_TL_DC_3RD_CLAMP.Error_T2.ATIME := T#0MS;
   S705_TL_DC_3RD_CLAMP.Adv_End_Aux := FALSE;
   S705_TL_DC_3RD_CLAMP.Ret_End_Aux := TRUE;
   S705_TL_DC_3RD_CLAMP.CHK_Aux1 := FALSE;
   S705_TL_DC_3RD_CLAMP.CHK_Aux2 := FALSE;
   S705_TL_DC_3RD_CLAMP.Error_T1_DN := FALSE;
   S705_TL_DC_3RD_CLAMP.Error_T2_DN := FALSE;
   S705_TL_DC_3RD_CLAMP.Adv_Memo := FALSE;
   S705_TL_DC_3RD_CLAMP.Visu_Adv_Arr[0] := FALSE;
   S705_TL_DC_3RD_CLAMP.Visu_Adv_Arr[1] := FALSE;
   S705_TL_DC_3RD_CLAMP.Visu_Adv_Arr[2] := FALSE;
   S705_TL_DC_3RD_CLAMP.Visu_Adv_Arr[3] := FALSE;
   S705_TL_DC_3RD_CLAMP.Visu_Adv_Arr[4] := FALSE;
   S705_TL_DC_3RD_CLAMP.Visu_Adv_Arr[5] := FALSE;
   S705_TL_DC_3RD_CLAMP.Visu_Adv_Arr[6] := FALSE;
   S705_TL_DC_3RD_CLAMP.Visu_Adv_Arr[7] := FALSE;
   S705_TL_DC_3RD_CLAMP.Visu_Adv_Arr[8] := FALSE;
   S705_TL_DC_3RD_CLAMP.Visu_Adv_Arr[9] := FALSE;
   S705_TL_DC_3RD_CLAMP.Visu_Adv_Arr[10] := FALSE;
   S705_TL_DC_3RD_CLAMP.Visu_Adv_Arr[11] := FALSE;
   S705_TL_DC_3RD_CLAMP.Visu_Adv_Arr[12] := FALSE;
   S705_TL_DC_3RD_CLAMP.Visu_Adv_Arr[13] := FALSE;
   S705_TL_DC_3RD_CLAMP.Visu_Adv_Arr[14] := FALSE;
   S705_TL_DC_3RD_CLAMP.Visu_Adv_Arr[15] := FALSE;
   S705_TL_DC_3RD_CLAMP.Visu_Ret_Arr[0] := TRUE;
   S705_TL_DC_3RD_CLAMP.Visu_Ret_Arr[1] := TRUE;
   S705_TL_DC_3RD_CLAMP.Visu_Ret_Arr[2] := FALSE;
   S705_TL_DC_3RD_CLAMP.Visu_Ret_Arr[3] := FALSE;
   S705_TL_DC_3RD_CLAMP.Visu_Ret_Arr[4] := FALSE;
   S705_TL_DC_3RD_CLAMP.Visu_Ret_Arr[5] := FALSE;
   S705_TL_DC_3RD_CLAMP.Visu_Ret_Arr[6] := FALSE;
   S705_TL_DC_3RD_CLAMP.Visu_Ret_Arr[7] := FALSE;
   S705_TL_DC_3RD_CLAMP.Visu_Ret_Arr[8] := FALSE;
   S705_TL_DC_3RD_CLAMP.Visu_Ret_Arr[9] := FALSE;
   S705_TL_DC_3RD_CLAMP.Visu_Ret_Arr[10] := FALSE;
   S705_TL_DC_3RD_CLAMP.Visu_Ret_Arr[11] := FALSE;
   S705_TL_DC_3RD_CLAMP.Visu_Ret_Arr[12] := FALSE;
   S705_TL_DC_3RD_CLAMP.Visu_Ret_Arr[13] := FALSE;
   S705_TL_DC_3RD_CLAMP.Visu_Ret_Arr[14] := FALSE;
   S705_TL_DC_3RD_CLAMP.Visu_Ret_Arr[15] := FALSE;
   S705_TL_DC_3RD_CLAMP.BLK_Move_Ret := 0;
   S705_TL_DC_3RD_CLAMP.Enable := TRUE;
   S705_TL_DC_3RD_CLAMP.Adv_End := FALSE;
   S705_TL_DC_3RD_CLAMP.Ret_End := TRUE;
   S705_TL_DC_U262_1_UP_DN.Enable_Aux := TRUE;
   S705_TL_DC_U262_1_UP_DN.Adv_Amount := 1;
   S705_TL_DC_U262_1_UP_DN.Ret_Amount := 1;
   S705_TL_DC_U262_1_UP_DN.LS_Adv1 := FALSE;
   S705_TL_DC_U262_1_UP_DN.LS_Ret1 := TRUE;
   S705_TL_DC_U262_1_UP_DN.LS_Adv2 := FALSE;
   S705_TL_DC_U262_1_UP_DN.LS_Ret2 := FALSE;
   S705_TL_DC_U262_1_UP_DN.LS_Adv3 := FALSE;
   S705_TL_DC_U262_1_UP_DN.LS_Ret3 := FALSE;
   S705_TL_DC_U262_1_UP_DN.LS_Adv4 := FALSE;
   S705_TL_DC_U262_1_UP_DN.LS_Ret4 := FALSE;
   S705_TL_DC_U262_1_UP_DN.LS_Adv5 := FALSE;
   S705_TL_DC_U262_1_UP_DN.LS_Ret5 := FALSE;
   S705_TL_DC_U262_1_UP_DN.LS_Adv6 := FALSE;
   S705_TL_DC_U262_1_UP_DN.LS_Ret6 := FALSE;
   S705_TL_DC_U262_1_UP_DN.LS_Adv7 := FALSE;
   S705_TL_DC_U262_1_UP_DN.LS_Ret7 := FALSE;
   S705_TL_DC_U262_1_UP_DN.LS_Adv8 := FALSE;
   S705_TL_DC_U262_1_UP_DN.LS_Ret8 := FALSE;
   S705_TL_DC_U262_1_UP_DN.SOL_Adv := FALSE;
   S705_TL_DC_U262_1_UP_DN.SOL_Ret := FALSE;
   S705_TL_DC_U262_1_UP_DN.M_Ready := TRUE;
   S705_TL_DC_U262_1_UP_DN.T_CHK1 := T#4S;
   S705_TL_DC_U262_1_UP_DN.T_CHK2 := T#4S;
   S705_TL_DC_U262_1_UP_DN.PB_Lamp_CHK := FALSE;
   S705_TL_DC_U262_1_UP_DN.PB_Error_Rst := FALSE;
   S705_TL_DC_U262_1_UP_DN.M_FLICK := TRUE;
   S705_TL_DC_U262_1_UP_DN.M_Adv_Err := FALSE;
   S705_TL_DC_U262_1_UP_DN.M_Ret_Err := FALSE;
   S705_TL_DC_U262_1_UP_DN.LP_Adv := FALSE;
   S705_TL_DC_U262_1_UP_DN.LP_Ret := TRUE;
   S705_TL_DC_U262_1_UP_DN.Visu_Adv := W#16#0;
   S705_TL_DC_U262_1_UP_DN.Visu_Ret := W#16#300;
   S705_TL_DC_U262_1_UP_DN.Error_T1.IN := FALSE;
   S705_TL_DC_U262_1_UP_DN.Error_T1.PT := T#4S;
   S705_TL_DC_U262_1_UP_DN.Error_T1.Q := FALSE;
   S705_TL_DC_U262_1_UP_DN.Error_T1.ET := T#0MS;
   S705_TL_DC_U262_1_UP_DN.Error_T1.STATE := B#16#0;
   S705_TL_DC_U262_1_UP_DN.Error_T1.STIME := T#23D5H8M46S916MS;
   S705_TL_DC_U262_1_UP_DN.Error_T1.ATIME := T#23D5H8M46S961MS;
   S705_TL_DC_U262_1_UP_DN.Error_T2.IN := FALSE;
   S705_TL_DC_U262_1_UP_DN.Error_T2.PT := T#4S;
   S705_TL_DC_U262_1_UP_DN.Error_T2.Q := FALSE;
   S705_TL_DC_U262_1_UP_DN.Error_T2.ET := T#0MS;
   S705_TL_DC_U262_1_UP_DN.Error_T2.STATE := B#16#0;
   S705_TL_DC_U262_1_UP_DN.Error_T2.STIME := T#0MS;
   S705_TL_DC_U262_1_UP_DN.Error_T2.ATIME := T#0MS;
   S705_TL_DC_U262_1_UP_DN.Adv_End_Aux := FALSE;
   S705_TL_DC_U262_1_UP_DN.Ret_End_Aux := TRUE;
   S705_TL_DC_U262_1_UP_DN.CHK_Aux1 := FALSE;
   S705_TL_DC_U262_1_UP_DN.CHK_Aux2 := FALSE;
   S705_TL_DC_U262_1_UP_DN.Error_T1_DN := FALSE;
   S705_TL_DC_U262_1_UP_DN.Error_T2_DN := FALSE;
   S705_TL_DC_U262_1_UP_DN.Adv_Memo := FALSE;
   S705_TL_DC_U262_1_UP_DN.Visu_Adv_Arr[0] := FALSE;
   S705_TL_DC_U262_1_UP_DN.Visu_Adv_Arr[1] := FALSE;
   S705_TL_DC_U262_1_UP_DN.Visu_Adv_Arr[2] := FALSE;
   S705_TL_DC_U262_1_UP_DN.Visu_Adv_Arr[3] := FALSE;
   S705_TL_DC_U262_1_UP_DN.Visu_Adv_Arr[4] := FALSE;
   S705_TL_DC_U262_1_UP_DN.Visu_Adv_Arr[5] := FALSE;
   S705_TL_DC_U262_1_UP_DN.Visu_Adv_Arr[6] := FALSE;
   S705_TL_DC_U262_1_UP_DN.Visu_Adv_Arr[7] := FALSE;
   S705_TL_DC_U262_1_UP_DN.Visu_Adv_Arr[8] := FALSE;
   S705_TL_DC_U262_1_UP_DN.Visu_Adv_Arr[9] := FALSE;
   S705_TL_DC_U262_1_UP_DN.Visu_Adv_Arr[10] := FALSE;
   S705_TL_DC_U262_1_UP_DN.Visu_Adv_Arr[11] := FALSE;
   S705_TL_DC_U262_1_UP_DN.Visu_Adv_Arr[12] := FALSE;
   S705_TL_DC_U262_1_UP_DN.Visu_Adv_Arr[13] := FALSE;
   S705_TL_DC_U262_1_UP_DN.Visu_Adv_Arr[14] := FALSE;
   S705_TL_DC_U262_1_UP_DN.Visu_Adv_Arr[15] := FALSE;
   S705_TL_DC_U262_1_UP_DN.Visu_Ret_Arr[0] := TRUE;
   S705_TL_DC_U262_1_UP_DN.Visu_Ret_Arr[1] := TRUE;
   S705_TL_DC_U262_1_UP_DN.Visu_Ret_Arr[2] := FALSE;
   S705_TL_DC_U262_1_UP_DN.Visu_Ret_Arr[3] := FALSE;
   S705_TL_DC_U262_1_UP_DN.Visu_Ret_Arr[4] := FALSE;
   S705_TL_DC_U262_1_UP_DN.Visu_Ret_Arr[5] := FALSE;
   S705_TL_DC_U262_1_UP_DN.Visu_Ret_Arr[6] := FALSE;
   S705_TL_DC_U262_1_UP_DN.Visu_Ret_Arr[7] := FALSE;
   S705_TL_DC_U262_1_UP_DN.Visu_Ret_Arr[8] := FALSE;
   S705_TL_DC_U262_1_UP_DN.Visu_Ret_Arr[9] := FALSE;
   S705_TL_DC_U262_1_UP_DN.Visu_Ret_Arr[10] := FALSE;
   S705_TL_DC_U262_1_UP_DN.Visu_Ret_Arr[11] := FALSE;
   S705_TL_DC_U262_1_UP_DN.Visu_Ret_Arr[12] := FALSE;
   S705_TL_DC_U262_1_UP_DN.Visu_Ret_Arr[13] := FALSE;
   S705_TL_DC_U262_1_UP_DN.Visu_Ret_Arr[14] := FALSE;
   S705_TL_DC_U262_1_UP_DN.Visu_Ret_Arr[15] := FALSE;
   S705_TL_DC_U262_1_UP_DN.BLK_Move_Ret := 0;
   S705_TL_DC_U262_1_UP_DN.Enable := TRUE;
   S705_TL_DC_U262_1_UP_DN.Adv_End := FALSE;
   S705_TL_DC_U262_1_UP_DN.Ret_End := TRUE;
   S705_TL_DC_U262_1.Enable_Aux := TRUE;
   S705_TL_DC_U262_1.Adv_Amount := 1;
   S705_TL_DC_U262_1.Ret_Amount := 1;
   S705_TL_DC_U262_1.LS_Adv1 := FALSE;
   S705_TL_DC_U262_1.LS_Ret1 := TRUE;
   S705_TL_DC_U262_1.LS_Adv2 := FALSE;
   S705_TL_DC_U262_1.LS_Ret2 := FALSE;
   S705_TL_DC_U262_1.LS_Adv3 := FALSE;
   S705_TL_DC_U262_1.LS_Ret3 := FALSE;
   S705_TL_DC_U262_1.LS_Adv4 := FALSE;
   S705_TL_DC_U262_1.LS_Ret4 := FALSE;
   S705_TL_DC_U262_1.LS_Adv5 := FALSE;
   S705_TL_DC_U262_1.LS_Ret5 := FALSE;
   S705_TL_DC_U262_1.LS_Adv6 := FALSE;
   S705_TL_DC_U262_1.LS_Ret6 := FALSE;
   S705_TL_DC_U262_1.LS_Adv7 := FALSE;
   S705_TL_DC_U262_1.LS_Ret7 := FALSE;
   S705_TL_DC_U262_1.LS_Adv8 := FALSE;
   S705_TL_DC_U262_1.LS_Ret8 := FALSE;
   S705_TL_DC_U262_1.SOL_Adv := FALSE;
   S705_TL_DC_U262_1.SOL_Ret := FALSE;
   S705_TL_DC_U262_1.M_Ready := TRUE;
   S705_TL_DC_U262_1.T_CHK1 := T#4S;
   S705_TL_DC_U262_1.T_CHK2 := T#4S;
   S705_TL_DC_U262_1.PB_Lamp_CHK := FALSE;
   S705_TL_DC_U262_1.PB_Error_Rst := FALSE;
   S705_TL_DC_U262_1.M_FLICK := TRUE;
   S705_TL_DC_U262_1.M_Adv_Err := FALSE;
   S705_TL_DC_U262_1.M_Ret_Err := FALSE;
   S705_TL_DC_U262_1.LP_Adv := FALSE;
   S705_TL_DC_U262_1.LP_Ret := TRUE;
   S705_TL_DC_U262_1.Visu_Adv := W#16#0;
   S705_TL_DC_U262_1.Visu_Ret := W#16#300;
   S705_TL_DC_U262_1.Error_T1.IN := FALSE;
   S705_TL_DC_U262_1.Error_T1.PT := T#4S;
   S705_TL_DC_U262_1.Error_T1.Q := FALSE;
   S705_TL_DC_U262_1.Error_T1.ET := T#0MS;
   S705_TL_DC_U262_1.Error_T1.STATE := B#16#0;
   S705_TL_DC_U262_1.Error_T1.STIME := T#23D5H8M46S916MS;
   S705_TL_DC_U262_1.Error_T1.ATIME := T#23D5H8M46S961MS;
   S705_TL_DC_U262_1.Error_T2.IN := FALSE;
   S705_TL_DC_U262_1.Error_T2.PT := T#4S;
   S705_TL_DC_U262_1.Error_T2.Q := FALSE;
   S705_TL_DC_U262_1.Error_T2.ET := T#0MS;
   S705_TL_DC_U262_1.Error_T2.STATE := B#16#0;
   S705_TL_DC_U262_1.Error_T2.STIME := T#0MS;
   S705_TL_DC_U262_1.Error_T2.ATIME := T#0MS;
   S705_TL_DC_U262_1.Adv_End_Aux := FALSE;
   S705_TL_DC_U262_1.Ret_End_Aux := TRUE;
   S705_TL_DC_U262_1.CHK_Aux1 := FALSE;
   S705_TL_DC_U262_1.CHK_Aux2 := FALSE;
   S705_TL_DC_U262_1.Error_T1_DN := FALSE;
   S705_TL_DC_U262_1.Error_T2_DN := FALSE;
   S705_TL_DC_U262_1.Adv_Memo := FALSE;
   S705_TL_DC_U262_1.Visu_Adv_Arr[0] := FALSE;
   S705_TL_DC_U262_1.Visu_Adv_Arr[1] := FALSE;
   S705_TL_DC_U262_1.Visu_Adv_Arr[2] := FALSE;
   S705_TL_DC_U262_1.Visu_Adv_Arr[3] := FALSE;
   S705_TL_DC_U262_1.Visu_Adv_Arr[4] := FALSE;
   S705_TL_DC_U262_1.Visu_Adv_Arr[5] := FALSE;
   S705_TL_DC_U262_1.Visu_Adv_Arr[6] := FALSE;
   S705_TL_DC_U262_1.Visu_Adv_Arr[7] := FALSE;
   S705_TL_DC_U262_1.Visu_Adv_Arr[8] := FALSE;
   S705_TL_DC_U262_1.Visu_Adv_Arr[9] := FALSE;
   S705_TL_DC_U262_1.Visu_Adv_Arr[10] := FALSE;
   S705_TL_DC_U262_1.Visu_Adv_Arr[11] := FALSE;
   S705_TL_DC_U262_1.Visu_Adv_Arr[12] := FALSE;
   S705_TL_DC_U262_1.Visu_Adv_Arr[13] := FALSE;
   S705_TL_DC_U262_1.Visu_Adv_Arr[14] := FALSE;
   S705_TL_DC_U262_1.Visu_Adv_Arr[15] := FALSE;
   S705_TL_DC_U262_1.Visu_Ret_Arr[0] := TRUE;
   S705_TL_DC_U262_1.Visu_Ret_Arr[1] := TRUE;
   S705_TL_DC_U262_1.Visu_Ret_Arr[2] := FALSE;
   S705_TL_DC_U262_1.Visu_Ret_Arr[3] := FALSE;
   S705_TL_DC_U262_1.Visu_Ret_Arr[4] := FALSE;
   S705_TL_DC_U262_1.Visu_Ret_Arr[5] := FALSE;
   S705_TL_DC_U262_1.Visu_Ret_Arr[6] := FALSE;
   S705_TL_DC_U262_1.Visu_Ret_Arr[7] := FALSE;
   S705_TL_DC_U262_1.Visu_Ret_Arr[8] := FALSE;
   S705_TL_DC_U262_1.Visu_Ret_Arr[9] := FALSE;
   S705_TL_DC_U262_1.Visu_Ret_Arr[10] := FALSE;
   S705_TL_DC_U262_1.Visu_Ret_Arr[11] := FALSE;
   S705_TL_DC_U262_1.Visu_Ret_Arr[12] := FALSE;
   S705_TL_DC_U262_1.Visu_Ret_Arr[13] := FALSE;
   S705_TL_DC_U262_1.Visu_Ret_Arr[14] := FALSE;
   S705_TL_DC_U262_1.Visu_Ret_Arr[15] := FALSE;
   S705_TL_DC_U262_1.BLK_Move_Ret := 0;
   S705_TL_DC_U262_1.Enable := TRUE;
   S705_TL_DC_U262_1.Adv_End := FALSE;
   S705_TL_DC_U262_1.Ret_End := TRUE;
   S705_TL_DC_U262_1_CLAMP.Enable_Aux := TRUE;
   S705_TL_DC_U262_1_CLAMP.Adv_Amount := 1;
   S705_TL_DC_U262_1_CLAMP.Ret_Amount := 1;
   S705_TL_DC_U262_1_CLAMP.LS_Adv1 := FALSE;
   S705_TL_DC_U262_1_CLAMP.LS_Ret1 := TRUE;
   S705_TL_DC_U262_1_CLAMP.LS_Adv2 := FALSE;
   S705_TL_DC_U262_1_CLAMP.LS_Ret2 := FALSE;
   S705_TL_DC_U262_1_CLAMP.LS_Adv3 := FALSE;
   S705_TL_DC_U262_1_CLAMP.LS_Ret3 := FALSE;
   S705_TL_DC_U262_1_CLAMP.LS_Adv4 := FALSE;
   S705_TL_DC_U262_1_CLAMP.LS_Ret4 := FALSE;
   S705_TL_DC_U262_1_CLAMP.LS_Adv5 := FALSE;
   S705_TL_DC_U262_1_CLAMP.LS_Ret5 := FALSE;
   S705_TL_DC_U262_1_CLAMP.LS_Adv6 := FALSE;
   S705_TL_DC_U262_1_CLAMP.LS_Ret6 := FALSE;
   S705_TL_DC_U262_1_CLAMP.LS_Adv7 := FALSE;
   S705_TL_DC_U262_1_CLAMP.LS_Ret7 := FALSE;
   S705_TL_DC_U262_1_CLAMP.LS_Adv8 := FALSE;
   S705_TL_DC_U262_1_CLAMP.LS_Ret8 := FALSE;
   S705_TL_DC_U262_1_CLAMP.SOL_Adv := FALSE;
   S705_TL_DC_U262_1_CLAMP.SOL_Ret := FALSE;
   S705_TL_DC_U262_1_CLAMP.M_Ready := TRUE;
   S705_TL_DC_U262_1_CLAMP.T_CHK1 := T#4S;
   S705_TL_DC_U262_1_CLAMP.T_CHK2 := T#4S;
   S705_TL_DC_U262_1_CLAMP.PB_Lamp_CHK := FALSE;
   S705_TL_DC_U262_1_CLAMP.PB_Error_Rst := FALSE;
   S705_TL_DC_U262_1_CLAMP.M_FLICK := TRUE;
   S705_TL_DC_U262_1_CLAMP.M_Adv_Err := FALSE;
   S705_TL_DC_U262_1_CLAMP.M_Ret_Err := FALSE;
   S705_TL_DC_U262_1_CLAMP.LP_Adv := FALSE;
   S705_TL_DC_U262_1_CLAMP.LP_Ret := TRUE;
   S705_TL_DC_U262_1_CLAMP.Visu_Adv := W#16#0;
   S705_TL_DC_U262_1_CLAMP.Visu_Ret := W#16#300;
   S705_TL_DC_U262_1_CLAMP.Error_T1.IN := FALSE;
   S705_TL_DC_U262_1_CLAMP.Error_T1.PT := T#4S;
   S705_TL_DC_U262_1_CLAMP.Error_T1.Q := FALSE;
   S705_TL_DC_U262_1_CLAMP.Error_T1.ET := T#0MS;
   S705_TL_DC_U262_1_CLAMP.Error_T1.STATE := B#16#0;
   S705_TL_DC_U262_1_CLAMP.Error_T1.STIME := T#23D5H8M46S916MS;
   S705_TL_DC_U262_1_CLAMP.Error_T1.ATIME := T#23D5H8M46S961MS;
   S705_TL_DC_U262_1_CLAMP.Error_T2.IN := FALSE;
   S705_TL_DC_U262_1_CLAMP.Error_T2.PT := T#4S;
   S705_TL_DC_U262_1_CLAMP.Error_T2.Q := FALSE;
   S705_TL_DC_U262_1_CLAMP.Error_T2.ET := T#0MS;
   S705_TL_DC_U262_1_CLAMP.Error_T2.STATE := B#16#0;
   S705_TL_DC_U262_1_CLAMP.Error_T2.STIME := T#0MS;
   S705_TL_DC_U262_1_CLAMP.Error_T2.ATIME := T#0MS;
   S705_TL_DC_U262_1_CLAMP.Adv_End_Aux := FALSE;
   S705_TL_DC_U262_1_CLAMP.Ret_End_Aux := TRUE;
   S705_TL_DC_U262_1_CLAMP.CHK_Aux1 := FALSE;
   S705_TL_DC_U262_1_CLAMP.CHK_Aux2 := FALSE;
   S705_TL_DC_U262_1_CLAMP.Error_T1_DN := FALSE;
   S705_TL_DC_U262_1_CLAMP.Error_T2_DN := FALSE;
   S705_TL_DC_U262_1_CLAMP.Adv_Memo := FALSE;
   S705_TL_DC_U262_1_CLAMP.Visu_Adv_Arr[0] := FALSE;
   S705_TL_DC_U262_1_CLAMP.Visu_Adv_Arr[1] := FALSE;
   S705_TL_DC_U262_1_CLAMP.Visu_Adv_Arr[2] := FALSE;
   S705_TL_DC_U262_1_CLAMP.Visu_Adv_Arr[3] := FALSE;
   S705_TL_DC_U262_1_CLAMP.Visu_Adv_Arr[4] := FALSE;
   S705_TL_DC_U262_1_CLAMP.Visu_Adv_Arr[5] := FALSE;
   S705_TL_DC_U262_1_CLAMP.Visu_Adv_Arr[6] := FALSE;
   S705_TL_DC_U262_1_CLAMP.Visu_Adv_Arr[7] := FALSE;
   S705_TL_DC_U262_1_CLAMP.Visu_Adv_Arr[8] := FALSE;
   S705_TL_DC_U262_1_CLAMP.Visu_Adv_Arr[9] := FALSE;
   S705_TL_DC_U262_1_CLAMP.Visu_Adv_Arr[10] := FALSE;
   S705_TL_DC_U262_1_CLAMP.Visu_Adv_Arr[11] := FALSE;
   S705_TL_DC_U262_1_CLAMP.Visu_Adv_Arr[12] := FALSE;
   S705_TL_DC_U262_1_CLAMP.Visu_Adv_Arr[13] := FALSE;
   S705_TL_DC_U262_1_CLAMP.Visu_Adv_Arr[14] := FALSE;
   S705_TL_DC_U262_1_CLAMP.Visu_Adv_Arr[15] := FALSE;
   S705_TL_DC_U262_1_CLAMP.Visu_Ret_Arr[0] := TRUE;
   S705_TL_DC_U262_1_CLAMP.Visu_Ret_Arr[1] := TRUE;
   S705_TL_DC_U262_1_CLAMP.Visu_Ret_Arr[2] := FALSE;
   S705_TL_DC_U262_1_CLAMP.Visu_Ret_Arr[3] := FALSE;
   S705_TL_DC_U262_1_CLAMP.Visu_Ret_Arr[4] := FALSE;
   S705_TL_DC_U262_1_CLAMP.Visu_Ret_Arr[5] := FALSE;
   S705_TL_DC_U262_1_CLAMP.Visu_Ret_Arr[6] := FALSE;
   S705_TL_DC_U262_1_CLAMP.Visu_Ret_Arr[7] := FALSE;
   S705_TL_DC_U262_1_CLAMP.Visu_Ret_Arr[8] := FALSE;
   S705_TL_DC_U262_1_CLAMP.Visu_Ret_Arr[9] := FALSE;
   S705_TL_DC_U262_1_CLAMP.Visu_Ret_Arr[10] := FALSE;
   S705_TL_DC_U262_1_CLAMP.Visu_Ret_Arr[11] := FALSE;
   S705_TL_DC_U262_1_CLAMP.Visu_Ret_Arr[12] := FALSE;
   S705_TL_DC_U262_1_CLAMP.Visu_Ret_Arr[13] := FALSE;
   S705_TL_DC_U262_1_CLAMP.Visu_Ret_Arr[14] := FALSE;
   S705_TL_DC_U262_1_CLAMP.Visu_Ret_Arr[15] := FALSE;
   S705_TL_DC_U262_1_CLAMP.BLK_Move_Ret := 0;
   S705_TL_DC_U262_1_CLAMP.Enable := TRUE;
   S705_TL_DC_U262_1_CLAMP.Adv_End := FALSE;
   S705_TL_DC_U262_1_CLAMP.Ret_End := TRUE;
   S705_TL_DC_U261_2_CLAMP.Enable_Aux := TRUE;
   S705_TL_DC_U261_2_CLAMP.Adv_Amount := 1;
   S705_TL_DC_U261_2_CLAMP.Ret_Amount := 1;
   S705_TL_DC_U261_2_CLAMP.LS_Adv1 := FALSE;
   S705_TL_DC_U261_2_CLAMP.LS_Ret1 := TRUE;
   S705_TL_DC_U261_2_CLAMP.LS_Adv2 := FALSE;
   S705_TL_DC_U261_2_CLAMP.LS_Ret2 := FALSE;
   S705_TL_DC_U261_2_CLAMP.LS_Adv3 := FALSE;
   S705_TL_DC_U261_2_CLAMP.LS_Ret3 := FALSE;
   S705_TL_DC_U261_2_CLAMP.LS_Adv4 := FALSE;
   S705_TL_DC_U261_2_CLAMP.LS_Ret4 := FALSE;
   S705_TL_DC_U261_2_CLAMP.LS_Adv5 := FALSE;
   S705_TL_DC_U261_2_CLAMP.LS_Ret5 := FALSE;
   S705_TL_DC_U261_2_CLAMP.LS_Adv6 := FALSE;
   S705_TL_DC_U261_2_CLAMP.LS_Ret6 := FALSE;
   S705_TL_DC_U261_2_CLAMP.LS_Adv7 := FALSE;
   S705_TL_DC_U261_2_CLAMP.LS_Ret7 := FALSE;
   S705_TL_DC_U261_2_CLAMP.LS_Adv8 := FALSE;
   S705_TL_DC_U261_2_CLAMP.LS_Ret8 := FALSE;
   S705_TL_DC_U261_2_CLAMP.SOL_Adv := FALSE;
   S705_TL_DC_U261_2_CLAMP.SOL_Ret := FALSE;
   S705_TL_DC_U261_2_CLAMP.M_Ready := TRUE;
   S705_TL_DC_U261_2_CLAMP.T_CHK1 := T#4S;
   S705_TL_DC_U261_2_CLAMP.T_CHK2 := T#4S;
   S705_TL_DC_U261_2_CLAMP.PB_Lamp_CHK := FALSE;
   S705_TL_DC_U261_2_CLAMP.PB_Error_Rst := FALSE;
   S705_TL_DC_U261_2_CLAMP.M_FLICK := TRUE;
   S705_TL_DC_U261_2_CLAMP.M_Adv_Err := FALSE;
   S705_TL_DC_U261_2_CLAMP.M_Ret_Err := FALSE;
   S705_TL_DC_U261_2_CLAMP.LP_Adv := FALSE;
   S705_TL_DC_U261_2_CLAMP.LP_Ret := TRUE;
   S705_TL_DC_U261_2_CLAMP.Visu_Adv := W#16#0;
   S705_TL_DC_U261_2_CLAMP.Visu_Ret := W#16#300;
   S705_TL_DC_U261_2_CLAMP.Error_T1.IN := FALSE;
   S705_TL_DC_U261_2_CLAMP.Error_T1.PT := T#4S;
   S705_TL_DC_U261_2_CLAMP.Error_T1.Q := FALSE;
   S705_TL_DC_U261_2_CLAMP.Error_T1.ET := T#0MS;
   S705_TL_DC_U261_2_CLAMP.Error_T1.STATE := B#16#0;
   S705_TL_DC_U261_2_CLAMP.Error_T1.STIME := T#23D5H8M46S916MS;
   S705_TL_DC_U261_2_CLAMP.Error_T1.ATIME := T#23D5H8M46S961MS;
   S705_TL_DC_U261_2_CLAMP.Error_T2.IN := FALSE;
   S705_TL_DC_U261_2_CLAMP.Error_T2.PT := T#4S;
   S705_TL_DC_U261_2_CLAMP.Error_T2.Q := FALSE;
   S705_TL_DC_U261_2_CLAMP.Error_T2.ET := T#0MS;
   S705_TL_DC_U261_2_CLAMP.Error_T2.STATE := B#16#0;
   S705_TL_DC_U261_2_CLAMP.Error_T2.STIME := T#0MS;
   S705_TL_DC_U261_2_CLAMP.Error_T2.ATIME := T#0MS;
   S705_TL_DC_U261_2_CLAMP.Adv_End_Aux := FALSE;
   S705_TL_DC_U261_2_CLAMP.Ret_End_Aux := TRUE;
   S705_TL_DC_U261_2_CLAMP.CHK_Aux1 := FALSE;
   S705_TL_DC_U261_2_CLAMP.CHK_Aux2 := FALSE;
   S705_TL_DC_U261_2_CLAMP.Error_T1_DN := FALSE;
   S705_TL_DC_U261_2_CLAMP.Error_T2_DN := FALSE;
   S705_TL_DC_U261_2_CLAMP.Adv_Memo := FALSE;
   S705_TL_DC_U261_2_CLAMP.Visu_Adv_Arr[0] := FALSE;
   S705_TL_DC_U261_2_CLAMP.Visu_Adv_Arr[1] := FALSE;
   S705_TL_DC_U261_2_CLAMP.Visu_Adv_Arr[2] := FALSE;
   S705_TL_DC_U261_2_CLAMP.Visu_Adv_Arr[3] := FALSE;
   S705_TL_DC_U261_2_CLAMP.Visu_Adv_Arr[4] := FALSE;
   S705_TL_DC_U261_2_CLAMP.Visu_Adv_Arr[5] := FALSE;
   S705_TL_DC_U261_2_CLAMP.Visu_Adv_Arr[6] := FALSE;
   S705_TL_DC_U261_2_CLAMP.Visu_Adv_Arr[7] := FALSE;
   S705_TL_DC_U261_2_CLAMP.Visu_Adv_Arr[8] := FALSE;
   S705_TL_DC_U261_2_CLAMP.Visu_Adv_Arr[9] := FALSE;
   S705_TL_DC_U261_2_CLAMP.Visu_Adv_Arr[10] := FALSE;
   S705_TL_DC_U261_2_CLAMP.Visu_Adv_Arr[11] := FALSE;
   S705_TL_DC_U261_2_CLAMP.Visu_Adv_Arr[12] := FALSE;
   S705_TL_DC_U261_2_CLAMP.Visu_Adv_Arr[13] := FALSE;
   S705_TL_DC_U261_2_CLAMP.Visu_Adv_Arr[14] := FALSE;
   S705_TL_DC_U261_2_CLAMP.Visu_Adv_Arr[15] := FALSE;
   S705_TL_DC_U261_2_CLAMP.Visu_Ret_Arr[0] := TRUE;
   S705_TL_DC_U261_2_CLAMP.Visu_Ret_Arr[1] := TRUE;
   S705_TL_DC_U261_2_CLAMP.Visu_Ret_Arr[2] := FALSE;
   S705_TL_DC_U261_2_CLAMP.Visu_Ret_Arr[3] := FALSE;
   S705_TL_DC_U261_2_CLAMP.Visu_Ret_Arr[4] := FALSE;
   S705_TL_DC_U261_2_CLAMP.Visu_Ret_Arr[5] := FALSE;
   S705_TL_DC_U261_2_CLAMP.Visu_Ret_Arr[6] := FALSE;
   S705_TL_DC_U261_2_CLAMP.Visu_Ret_Arr[7] := FALSE;
   S705_TL_DC_U261_2_CLAMP.Visu_Ret_Arr[8] := FALSE;
   S705_TL_DC_U261_2_CLAMP.Visu_Ret_Arr[9] := FALSE;
   S705_TL_DC_U261_2_CLAMP.Visu_Ret_Arr[10] := FALSE;
   S705_TL_DC_U261_2_CLAMP.Visu_Ret_Arr[11] := FALSE;
   S705_TL_DC_U261_2_CLAMP.Visu_Ret_Arr[12] := FALSE;
   S705_TL_DC_U261_2_CLAMP.Visu_Ret_Arr[13] := FALSE;
   S705_TL_DC_U261_2_CLAMP.Visu_Ret_Arr[14] := FALSE;
   S705_TL_DC_U261_2_CLAMP.Visu_Ret_Arr[15] := FALSE;
   S705_TL_DC_U261_2_CLAMP.BLK_Move_Ret := 0;
   S705_TL_DC_U261_2_CLAMP.Enable := TRUE;
   S705_TL_DC_U261_2_CLAMP.Adv_End := FALSE;
   S705_TL_DC_U261_2_CLAMP.Ret_End := TRUE;
END_DATA_BLOCK

FUNCTION FC 114 : VOID
TITLE =
VERSION : 0.1

BEGIN
NETWORK
TITLE =
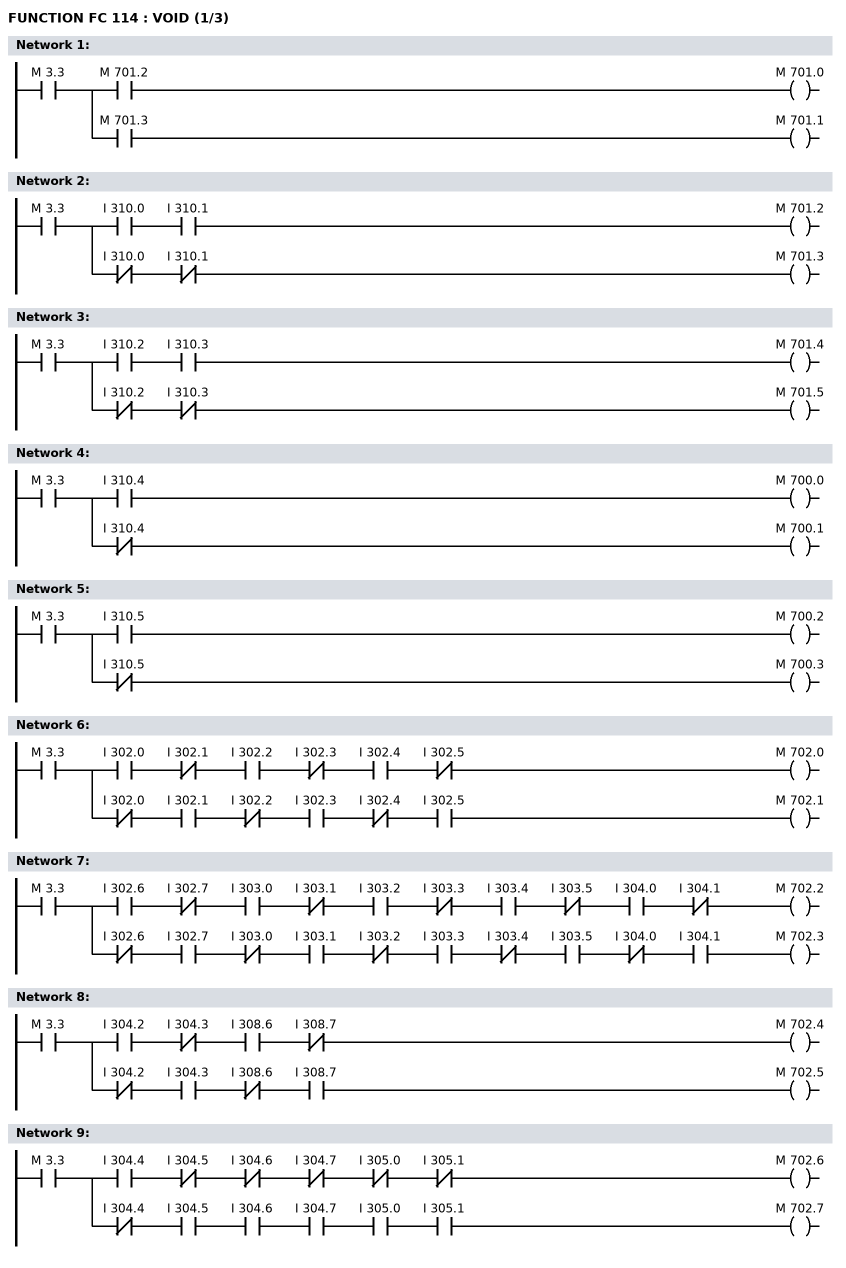

      A     M      3.3;
      =     L      0.0;
      A     L      0.0;
      A     M    701.2;
      =     M    701.0;
      A     L      0.0;
      A     M    701.3;
      =     M    701.1;
NETWORK
TITLE =

      A     M      3.3;
      =     L      0.0;
      A     L      0.0;
      A     I    310.0;
      A     I    310.1;
      =     M    701.2;
      A     L      0.0;
      AN    I    310.0;
      AN    I    310.1;
      =     M    701.3;
NETWORK
TITLE =

      A     M      3.3;
      =     L      0.0;
      A     L      0.0;
      A     I    310.2;
      A     I    310.3;
      =     M    701.4;
      A     L      0.0;
      AN    I    310.2;
      AN    I    310.3;
      =     M    701.5;
NETWORK
TITLE =

      A     M      3.3;
      =     L      0.0;
      A     L      0.0;
      A     I    310.4;
      =     M    700.0;
      A     L      0.0;
      AN    I    310.4;
      =     M    700.1;
NETWORK
TITLE =

      A     M      3.3;
      =     L      0.0;
      A     L      0.0;
      A     I    310.5;
      =     M    700.2;
      A     L      0.0;
      AN    I    310.5;
      =     M    700.3;
NETWORK
TITLE =

      A     M      3.3;
      =     L      0.0;
      A     L      0.0;
      A     I    302.0;
      AN    I    302.1;
      A     I    302.2;
      AN    I    302.3;
      A     I    302.4;
      AN    I    302.5;
      =     M    702.0;
      A     L      0.0;
      AN    I    302.0;
      A     I    302.1;
      AN    I    302.2;
      A     I    302.3;
      AN    I    302.4;
      A     I    302.5;
      =     M    702.1;
NETWORK
TITLE =

      A     M      3.3;
      =     L      0.0;
      A     L      0.0;
      A     I    302.6;
      AN    I    302.7;
      A     I    303.0;
      AN    I    303.1;
      A     I    303.2;
      AN    I    303.3;
      A     I    303.4;
      AN    I    303.5;
      A     I    304.0;
      AN    I    304.1;
      =     M    702.2;
      A     L      0.0;
      AN    I    302.6;
      A     I    302.7;
      AN    I    303.0;
      A     I    303.1;
      AN    I    303.2;
      A     I    303.3;
      AN    I    303.4;
      A     I    303.5;
      AN    I    304.0;
      A     I    304.1;
      =     M    702.3;
NETWORK
TITLE =

      A     M      3.3;
      =     L      0.0;
      A     L      0.0;
      A     I    304.2;
      AN    I    304.3;
      A     I    308.6;
      AN    I    308.7;
      =     M    702.4;
      A     L      0.0;
      AN    I    304.2;
      A     I    304.3;
      AN    I    308.6;
      A     I    308.7;
      =     M    702.5;
NETWORK
TITLE =

      A     M      3.3;
      =     L      0.0;
      A     L      0.0;
      A     I    304.4;
      AN    I    304.5;
      AN    I    304.6;
      AN    I    304.7;
      AN    I    305.0;
      AN    I    305.1;
      =     M    702.6;
      A     L      0.0;
      AN    I    304.4;
      A     I    304.5;
      A     I    304.6;
      A     I    304.7;
      A     I    305.0;
      A     I    305.1;
      =     M    702.7;
NETWORK
TITLE =
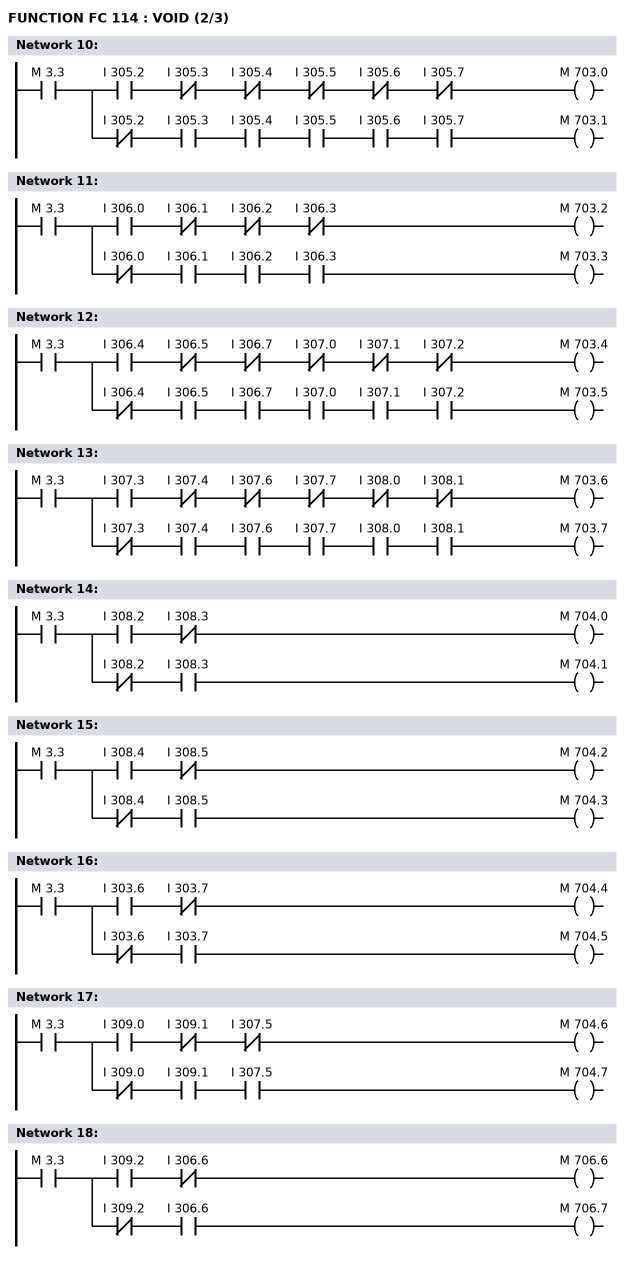

      A     M      3.3;
      =     L      0.0;
      A     L      0.0;
      A     I    305.2;
      AN    I    305.3;
      AN    I    305.4;
      AN    I    305.5;
      AN    I    305.6;
      AN    I    305.7;
      =     M    703.0;
      A     L      0.0;
      AN    I    305.2;
      A     I    305.3;
      A     I    305.4;
      A     I    305.5;
      A     I    305.6;
      A     I    305.7;
      =     M    703.1;
NETWORK
TITLE =

      A     M      3.3;
      =     L      0.0;
      A     L      0.0;
      A     I    306.0;
      AN    I    306.1;
      AN    I    306.2;
      AN    I    306.3;
      =     M    703.2;
      A     L      0.0;
      AN    I    306.0;
      A     I    306.1;
      A     I    306.2;
      A     I    306.3;
      =     M    703.3;
NETWORK
TITLE =

      A     M      3.3;
      =     L      0.0;
      A     L      0.0;
      A     I    306.4;
      AN    I    306.5;
      AN    I    306.7;
      AN    I    307.0;
      AN    I    307.1;
      AN    I    307.2;
      =     M    703.4;
      A     L      0.0;
      AN    I    306.4;
      A     I    306.5;
      A     I    306.7;
      A     I    307.0;
      A     I    307.1;
      A     I    307.2;
      =     M    703.5;
NETWORK
TITLE =

      A     M      3.3;
      =     L      0.0;
      A     L      0.0;
      A     I    307.3;
      AN    I    307.4;
      AN    I    307.6;
      AN    I    307.7;
      AN    I    308.0;
      AN    I    308.1;
      =     M    703.6;
      A     L      0.0;
      AN    I    307.3;
      A     I    307.4;
      A     I    307.6;
      A     I    307.7;
      A     I    308.0;
      A     I    308.1;
      =     M    703.7;
NETWORK
TITLE =

      A     M      3.3;
      =     L      0.0;
      A     L      0.0;
      A     I    308.2;
      AN    I    308.3;
      =     M    704.0;
      A     L      0.0;
      AN    I    308.2;
      A     I    308.3;
      =     M    704.1;
NETWORK
TITLE =

      A     M      3.3;
      =     L      0.0;
      A     L      0.0;
      A     I    308.4;
      AN    I    308.5;
      =     M    704.2;
      A     L      0.0;
      AN    I    308.4;
      A     I    308.5;
      =     M    704.3;
NETWORK
TITLE =

